Yaskawa INFORM job: DPRINT3D5.JBI

/JOB
//NAME DPRINT3D5
//POS
///NPOS 1005,0,0,0,0,0
///TOOL 9
///POSTYPE PULSE
///PULSE
C00000=38696,60824,-96309,77205,-122166,-85375,0
C00001=38701,60832,-96286,77203,-122174,-85369,0
C00002=38706,60841,-96263,77202,-122182,-85364,0
C00003=38711,60849,-96240,77201,-122190,-85358,0
C00004=38716,60857,-96218,77200,-122199,-85352,0
C00005=38721,60866,-96195,77199,-122207,-85346,0
C00006=38726,60874,-96172,77197,-122215,-85340,0
C00007=38731,60882,-96149,77196,-122223,-85334,0
C00008=38736,60891,-96126,77195,-122232,-85328,0
C00009=38741,60899,-96103,77194,-122240,-85322,0
C00010=38746,60907,-96080,77193,-122248,-85317,0
C00011=38751,60915,-96059,77191,-122256,-85311,0
C00012=38756,60922,-96038,77190,-122264,-85306,0
C00013=38761,60930,-96017,77188,-122272,-85300,0
C00014=38766,60938,-95996,77186,-122280,-85295,0
C00015=38771,60945,-95976,77185,-122289,-85290,0
C00016=38776,60953,-95954,77183,-122297,-85285,0
C00017=38796,60963,-95927,77168,-122315,-85279,0
C00018=38827,60979,-95885,77145,-122344,-85272,0
C00019=38858,60994,-95842,77121,-122374,-85264,0
C00020=38885,61007,-95807,77101,-122398,-85257,0
C00021=38908,61018,-95779,77083,-122418,-85253,0
C00022=38930,61028,-95751,77065,-122439,-85248,0
C00023=38951,61036,-95729,77049,-122456,-85245,0
C00024=38971,61044,-95708,77033,-122474,-85242,0
C00025=38991,61052,-95686,77017,-122491,-85238,0
C00026=39011,61060,-95664,77001,-122509,-85235,0
C00027=39031,61068,-95643,76985,-122526,-85231,0
C00028=39048,61074,-95626,76971,-122540,-85229,0
C00029=39065,61080,-95610,76957,-122555,-85227,0
C00030=39083,61086,-95594,76943,-122570,-85225,0
C00031=39100,61092,-95577,76928,-122584,-85223,0
C00032=39115,61097,-95565,76916,-122597,-85221,0
C00033=39130,61101,-95552,76903,-122609,-85220,0
C00034=39146,61106,-95540,76890,-122622,-85219,0
C00035=39161,61111,-95527,76877,-122633,-85217,0
C00036=39176,61115,-95515,76864,-122646,-85216,0
C00037=39192,61120,-95502,76851,-122659,-85214,0
C00038=39207,61125,-95490,76838,-122671,-85213,0
C00039=39221,61129,-95479,76826,-122683,-85212,0
C00040=39235,61132,-95469,76814,-122693,-85211,0
C00041=39249,61136,-95458,76803,-122705,-85210,0
C00042=39255,61133,-95467,76795,-122706,-85213,0
C00043=39268,61127,-95485,76780,-122710,-85220,0
C00044=39280,61120,-95503,76765,-122714,-85227,0
C00045=39293,61113,-95522,76749,-122717,-85235,0
C00046=39307,61106,-95543,76732,-122721,-85242,0
C00047=39320,61099,-95564,76715,-122724,-85250,0
C00048=39334,61091,-95584,76698,-122728,-85259,0
C00049=39348,61084,-95605,76682,-122732,-85266,0
C00050=39362,61076,-95625,76665,-122736,-85274,0
C00051=39375,61069,-95646,76648,-122739,-85282,0
C00052=39390,61061,-95669,76630,-122742,-85290,0
C00053=39405,61052,-95695,76611,-122746,-85300,0
C00054=39420,61042,-95720,76592,-122749,-85310,0
C00055=39436,61033,-95746,76572,-122753,-85320,0
C00056=39452,61023,-95775,76552,-122756,-85330,0
C00057=39470,61011,-95807,76529,-122760,-85342,0
C00058=39487,61000,-95839,76507,-122763,-85354,0
C00059=39504,60988,-95871,76485,-122765,-85365,0
C00060=39522,60977,-95903,76462,-122769,-85377,0
C00061=39540,60964,-95939,76438,-122772,-85390,0
C00062=39560,60950,-95978,76413,-122775,-85404,0
C00063=39579,60936,-96018,76387,-122777,-85418,0
C00064=39606,60914,-96077,76352,-122779,-85439,0
C00065=39632,60893,-96136,76316,-122782,-85460,0
C00066=39658,60872,-96194,76281,-122784,-85481,0
C00067=39670,60862,-96222,76264,-122785,-85490,0
C00068=39672,60858,-96233,76261,-122783,-85494,0
C00069=39674,60850,-96255,76255,-122779,-85501,0
C00070=39677,60843,-96276,76249,-122776,-85507,0
C00071=39680,60835,-96298,76242,-122772,-85513,0
C00072=39682,60827,-96320,76236,-122769,-85520,0
C00073=39685,60818,-96343,76230,-122764,-85527,0
C00074=39687,60809,-96369,76223,-122761,-85535,0
C00075=39690,60800,-96394,76216,-122756,-85542,0
C00076=39693,60791,-96419,76210,-122752,-85550,0
C00077=39695,60782,-96444,76203,-122747,-85558,0
C00078=39698,60773,-96469,76196,-122742,-85566,0
C00079=39701,60764,-96495,76189,-122738,-85573,0
C00080=39703,60757,-96514,76183,-122736,-85579,0
C00081=39706,60749,-96536,76177,-122732,-85586,0
C00082=39709,60740,-96561,76170,-122728,-85593,0
C00083=39712,60731,-96586,76163,-122723,-85601,0
C00084=39715,60722,-96610,76157,-122719,-85608,0
C00085=39717,60713,-96635,76150,-122715,-85616,0
C00086=39720,60705,-96659,76144,-122710,-85623,0
C00087=39722,60696,-96683,76137,-122706,-85631,0
C00088=39725,60686,-96709,76131,-122701,-85638,0
C00089=39727,60677,-96735,76124,-122696,-85646,0
C00090=39729,60668,-96761,76117,-122692,-85654,0
C00091=39732,60658,-96787,76111,-122687,-85661,0
C00092=39734,60649,-96813,76104,-122683,-85669,0
C00093=39737,60640,-96839,76097,-122678,-85677,0
C00094=39739,60630,-96865,76091,-122674,-85685,0
C00095=39742,60621,-96891,76084,-122669,-85693,0
C00096=39744,60612,-96917,76077,-122663,-85701,0
C00097=39756,60552,-97082,76038,-122631,-85749,0
C00098=39779,60443,-97386,75966,-122571,-85840,0
C00099=39801,60334,-97689,75895,-122511,-85931,0
C00100=37705,58030,-104183,76996,-119736,-87530,0
C00101=42893,55575,-111597,70566,-120383,-90390,0
C00102=44083,55092,-113117,69083,-120456,-90996,0
C00103=26168,57356,-105949,67419,-123808,-89301,0
C00104=27034,56626,-108119,66140,-123522,-90049,0
C00105=31953,53610,-117563,59303,-122121,-93446,0
C00106=30382,53758,-117056,61107,-121729,-93060,0
C00107=38783,58034,-104194,75907,-120329,-87674,0
C00108=39450,58029,-104221,75227,-120689,-87771,0
C00109=39922,58098,-104031,74776,-120996,-87780,0
C00110=45754,54027,-116526,66798,-120045,-92214,0
C00111=45628,53809,-117229,66835,-119751,-92400,0
C00112=45552,53437,-118440,66749,-119301,-92742,0
C00113=45617,53075,-119644,66515,-118904,-93101,0
C00114=45741,52870,-120334,66287,-118707,-93318,0
C00115=31651,54009,-116270,59832,-122529,-93048,0
C00116=31289,54125,-115889,60288,-122540,-92886,0
C00117=30631,54256,-115460,61077,-122448,-92662,0
C00118=30631,54197,-115483,61087,-122475,-92644,0
C00119=46744,53849,-116954,65681,-120330,-92450,0
C00120=46504,53563,-117878,65809,-119907,-92681,0
C00121=46379,53276,-118815,65814,-119525,-92934,0
C00122=46365,52987,-119775,65696,-119175,-93211,0
C00123=46470,52706,-120722,65455,-118871,-93500,0
C00124=46705,52431,-121665,65073,-118611,-93804,0
C00125=31523,53166,-118835,59604,-121482,-93698,0
C00126=31058,53355,-118207,60207,-121566,-93455,0
C00127=30557,53489,-117756,60825,-121555,-93254,0
C00128=30011,53574,-117472,61466,-121459,-93092,0
C00129=29441,53602,-117370,62104,-121278,-92977,0
C00130=28834,53572,-117459,62754,-121010,-92911,0
C00131=24589,59209,-100464,70024,-124680,-87478,0
C00132=24940,59524,-99580,69821,-125135,-87290,0
C00133=25186,59870,-98613,69744,-125558,-87061,0
C00134=25338,60251,-97555,69782,-125954,-86793,0
C00135=25398,60656,-96433,69931,-126315,-86491,0
C00136=29543,55041,-112814,84218,-113592,-89272,0
C00137=37638,58636,-102304,77346,-120164,-86947,0
C00138=38105,58441,-102870,76796,-120296,-87172,0
C00139=38585,58332,-103192,76267,-120488,-87330,0
C00140=39084,58302,-103290,75750,-120742,-87425,0
C00141=39577,58348,-103167,75271,-121047,-87456,0
C00142=40060,58474,-102816,74836,-121406,-87421,0
C00143=46673,53886,-116833,65775,-120344,-92405,0
C00144=47998,53898,-116829,64338,-120877,-92595,0
C00145=47754,53769,-117239,64544,-120631,-92676,0
C00146=47542,53605,-117768,64698,-120356,-92795,0
C00147=47392,53423,-118360,64776,-120082,-92943,0
C00148=47314,53230,-118990,64773,-119821,-93113,0
C00149=47311,53035,-119640,64686,-119581,-93299,0
C00150=47388,52844,-120280,64514,-119373,-93493,0
C00151=47544,52667,-120884,64261,-119205,-93688,0
C00152=47774,52509,-121426,63936,-119085,-93874,0
C00153=47986,52416,-121752,63661,-119035,-93996,0
C00154=31245,52544,-120910,59613,-120533,-94224,0
C00155=31075,52695,-120397,59873,-120683,-94058,0
C00156=30835,52836,-119918,60205,-120793,-93891,0
C00157=30537,52956,-119514,60592,-120849,-93735,0
C00158=30196,53045,-119210,61010,-120845,-93600,0
C00159=29822,53102,-119017,61448,-120783,-93491,0
C00160=29430,53120,-118948,61887,-120665,-93414,0
C00161=29034,53101,-119004,62313,-120495,-93372,0
C00162=28650,53044,-119187,62707,-120280,-93368,0
C00163=28393,52977,-119404,62957,-120101,-93393,0
C00164=23585,59460,-99742,71179,-124323,-87108,0
C00165=23807,59542,-99515,70991,-124513,-87081,0
C00166=24080,59704,-99065,70793,-124797,-86999,0
C00167=24304,59906,-98501,70665,-125087,-86879,0
C00168=24472,60142,-97846,70612,-125369,-86724,0
C00169=24578,60399,-97134,70634,-125635,-86543,0
C00170=24622,60672,-96378,70729,-125875,-86339,0
C00171=24602,60947,-95620,70890,-126076,-86124,0
C00172=24522,61212,-94891,71108,-126232,-85906,0
C00173=24397,61437,-94275,71349,-126328,-85711,0
C00174=37719,59468,-99947,77613,-120758,-86270,0
C00175=37870,59314,-100383,77399,-120746,-86417,0
C00176=38128,59141,-100876,77070,-120782,-86594,0
C00177=38423,59016,-101237,76721,-120867,-86739,0
C00178=38744,58942,-101455,76368,-120999,-86845,0
C00179=39075,58921,-101521,76027,-121174,-86909,0
C00180=39402,58952,-101438,75712,-121381,-86930,0
C00181=39712,59035,-101210,75436,-121615,-86908,0
C00182=39992,59164,-100849,75212,-121866,-86843,0
C00183=40209,59320,-100413,75063,-122100,-86749,0
C00184=47926,53934,-116712,64434,-120891,-92551,0
C00185=48152,53085,-119498,63788,-119950,-93374,0
C00186=48199,52975,-119865,63685,-119829,-93485,0
C00187=48291,52871,-120214,63535,-119731,-93598,0
C00188=48427,52779,-120528,63344,-119660,-93706,0
C00189=48601,52701,-120797,63115,-119621,-93806,0
C00190=48757,52657,-120952,62923,-119617,-93872,0
C00191=48850,52637,-121023,62812,-119622,-93905,0
C00192=49432,52574,-121252,62141,-119740,-94050,0
C00193=30479,51877,-123192,60148,-119327,-94748,0
C00194=30570,52120,-122347,60161,-119708,-94525,0
C00195=30564,52217,-122016,60212,-119842,-94432,0
C00196=30517,52310,-121692,60308,-119958,-94335,0
C00197=30474,52355,-121539,60377,-120006,-94287,0
C00198=30461,52376,-121467,60401,-120032,-94265,0
C00199=30361,52466,-121160,60553,-120121,-94165,0
C00200=30228,52544,-120892,60737,-120183,-94072,0
C00201=30060,52610,-120664,60954,-120215,-93983,0
C00202=29864,52661,-120490,61193,-120215,-93907,0
C00203=29649,52692,-120380,61445,-120182,-93845,0
C00204=29420,52703,-120340,61701,-120115,-93802,0
C00205=29188,52692,-120373,61952,-120018,-93778,0
C00206=28961,52659,-120480,62186,-119894,-93776,0
C00207=28747,52604,-120659,62396,-119747,-93797,0
C00208=28604,52549,-120844,62527,-119622,-93829,0
C00209=28531,52514,-120960,62591,-119551,-93852,0
C00210=28194,52279,-121756,62854,-119121,-94032,0
C00211=22562,59976,-98286,72468,-124138,-86531,0
C00212=22998,59940,-98389,72010,-124363,-86630,0
C00213=23084,59942,-98387,71924,-124413,-86644,0
C00214=23278,59978,-98289,71744,-124554,-86648,0
C00215=23458,60045,-98105,71595,-124709,-86626,0
C00216=23615,60139,-97843,71482,-124874,-86578,0
C00217=23745,60257,-97517,71409,-125040,-86508,0
C00218=23842,60393,-97142,71379,-125202,-86419,0
C00219=23904,60539,-96737,71389,-125351,-86316,0
C00220=23931,60694,-96309,71440,-125485,-86200,0
C00221=23922,60848,-95885,71527,-125597,-86080,0
C00222=23879,60995,-95479,71645,-125683,-85958,0
C00223=23842,61062,-95294,71716,-125712,-85900,0
C00224=23830,61094,-95206,71744,-125729,-85874,0
C00225=23751,61224,-94850,71890,-125777,-85760,0
C00226=23644,61337,-94538,72054,-125798,-85654,0
C00227=23516,61430,-94282,72230,-125788,-85560,0
C00228=23138,61610,-93787,72697,-125688,-85357,0
C00229=38077,60419,-97294,77668,-121580,-85549,0
C00230=38146,60056,-98304,77443,-121390,-85850,0
C00231=38169,59988,-98497,77391,-121360,-85910,0
C00232=38258,59841,-98908,77239,-121319,-86041,0
C00233=38381,59715,-99264,77063,-121308,-86160,0
C00234=38530,59614,-99551,76871,-121330,-86264,0
C00235=38700,59541,-99759,76672,-121381,-86348,0
C00236=38881,59498,-99884,76472,-121458,-86409,0
C00237=39067,59486,-99921,76281,-121558,-86445,0
C00238=39250,59504,-99874,76107,-121676,-86457,0
C00239=39422,59551,-99746,75956,-121808,-86445,0
C00240=39576,59623,-99546,75833,-121947,-86408,0
C00241=39644,59672,-99411,75788,-122020,-86379,0
C00242=39678,59691,-99357,75762,-122053,-86369,0
C00243=39796,59787,-99091,75687,-122187,-86309,0
C00244=39892,59903,-98766,75644,-122324,-86229,0
C00245=39958,60034,-98403,75637,-122453,-86134,0
C00246=40046,60396,-97396,75714,-122752,-85858,0
C00247=49524,53763,-117308,62604,-121298,-92956,0
C00248=49011,53716,-117445,63144,-121047,-92918,0
C00249=48822,53679,-117560,63333,-120931,-92922,0
C00250=48650,53624,-117734,63495,-120799,-92946,0
C00251=48575,53588,-117849,63561,-120727,-92967,0
C00252=48537,53575,-117892,63595,-120697,-92974,0
C00253=48391,53498,-118139,63720,-120549,-93023,0
C00254=48274,53407,-118435,63805,-120394,-93089,0
C00255=48192,53305,-118769,63847,-120237,-93172,0
C00256=48150,53196,-119127,63842,-120088,-93269,0
C00257=48151,53135,-119329,63812,-120012,-93326,0
C00258=47967,53016,-119720,63958,-119797,-93412,0
C00259=49473,53563,-117956,62563,-121031,-93129,0
C00260=49558,53551,-117998,62464,-121049,-93154,0
C00261=49728,53527,-118081,62266,-121081,-93202,0
C00262=49820,53514,-118126,62159,-121098,-93229,0
C00263=49833,53512,-118134,62143,-121100,-93233,0
C00264=49848,53510,-118141,62126,-121103,-93237,0
C00265=49863,53508,-118148,62109,-121106,-93241,0
C00266=49878,53506,-118155,62091,-121110,-93245,0
C00267=49894,53504,-118161,62073,-121112,-93249,0
C00268=49909,53502,-118168,62055,-121115,-93253,0
C00269=49924,53500,-118175,62037,-121119,-93258,0
C00270=49937,53498,-118181,62022,-121121,-93262,0
C00271=49950,53496,-118188,62007,-121123,-93266,0
C00272=49963,53494,-118195,61992,-121126,-93269,0
C00273=49976,53492,-118203,61977,-121128,-93273,0
C00274=49988,53490,-118210,61962,-121129,-93277,0
C00275=50001,53488,-118218,61947,-121130,-93281,0
C00276=50014,53485,-118226,61932,-121132,-93285,0
C00277=50026,53483,-118234,61917,-121134,-93289,0
C00278=50039,53481,-118242,61902,-121136,-93294,0
C00279=50052,53479,-118249,61887,-121137,-93298,0
C00280=50064,53476,-118257,61872,-121139,-93302,0
C00281=50077,53474,-118265,61857,-121141,-93306,0
C00282=50090,53472,-118273,61842,-121143,-93310,0
C00283=50102,53469,-118281,61827,-121144,-93314,0
C00284=50115,53467,-118288,61812,-121146,-93318,0
C00285=50126,53465,-118296,61799,-121147,-93322,0
C00286=50136,53463,-118304,61786,-121149,-93325,0
C00287=50147,53460,-118312,61773,-121150,-93330,0
C00288=50158,53458,-118319,61760,-121150,-93333,0
C00289=50169,53456,-118327,61747,-121151,-93337,0
C00290=50179,53454,-118335,61734,-121152,-93341,0
C00291=50190,53451,-118342,61722,-121153,-93344,0
C00292=50199,53449,-118350,61710,-121153,-93348,0
C00293=50209,53447,-118358,61698,-121154,-93352,0
C00294=50219,53444,-118366,61686,-121154,-93356,0
C00295=50229,53442,-118375,61674,-121155,-93359,0
C00296=50239,53440,-118383,61662,-121155,-93363,0
C00297=50262,53425,-118431,61630,-121146,-93379,0
C00298=50284,53411,-118478,61598,-121136,-93396,0
C00299=50304,53398,-118520,61570,-121127,-93411,0
C00300=50320,53387,-118557,61547,-121118,-93424,0
C00301=50336,53376,-118595,61524,-121110,-93436,0
C00302=50351,53365,-118630,61502,-121101,-93448,0
C00303=50364,53356,-118662,61484,-121093,-93459,0
C00304=50376,53346,-118694,61465,-121085,-93470,0
C00305=50389,53336,-118727,61447,-121077,-93481,0
C00306=50402,53327,-118759,61428,-121069,-93491,0
C00307=50414,53317,-118792,61409,-121061,-93502,0
C00308=50427,53307,-118824,61391,-121053,-93513,0
C00309=50437,53299,-118851,61376,-121045,-93523,0
C00310=50447,53290,-118880,61361,-121038,-93532,0
C00311=50457,53282,-118908,61346,-121030,-93541,0
C00312=50467,53273,-118936,61331,-121023,-93551,0
C00313=50477,53265,-118964,61316,-121015,-93560,0
C00314=50484,53258,-118988,61304,-121010,-93567,0
C00315=50481,53254,-119001,61305,-121004,-93571,0
C00316=50477,53246,-119027,61307,-120991,-93577,0
C00317=50472,53238,-119054,61308,-120979,-93584,0
C00318=50467,53230,-119080,61310,-120967,-93591,0
C00319=50462,53222,-119107,61312,-120954,-93597,0
C00320=50457,53214,-119133,61313,-120942,-93604,0
C00321=50452,53206,-119159,61315,-120930,-93610,0
C00322=50447,53198,-119186,61317,-120918,-93617,0
C00323=50442,53190,-119212,61318,-120905,-93624,0
C00324=50436,53182,-119240,61321,-120892,-93630,0
C00325=50429,53173,-119267,61324,-120879,-93637,0
C00326=50423,53165,-119296,61327,-120866,-93644,0
C00327=50417,53156,-119324,61329,-120852,-93651,0
C00328=50411,53148,-119351,61332,-120839,-93658,0
C00329=50403,53138,-119383,61337,-120823,-93665,0
C00330=50394,53128,-119416,61341,-120807,-93673,0
C00331=50386,53118,-119448,61346,-120792,-93681,0
C00332=50378,53109,-119480,61350,-120776,-93689,0
C00333=50369,53099,-119512,61355,-120760,-93696,0
C00334=50361,53089,-119544,61359,-120745,-93704,0
C00335=50353,53080,-119575,61364,-120729,-93711,0
C00336=50343,53070,-119610,61369,-120713,-93719,0
C00337=50333,53059,-119645,61376,-120695,-93728,0
C00338=50322,53048,-119681,61382,-120676,-93736,0
C00339=50309,53036,-119721,61391,-120656,-93746,0
C00340=50294,53022,-119766,61401,-120633,-93756,0
C00341=50279,53008,-119812,61412,-120608,-93766,0
C00342=50263,52995,-119858,61422,-120585,-93777,0
C00343=50248,52981,-119903,61432,-120563,-93787,0
C00344=50229,52965,-119955,61445,-120535,-93799,0
C00345=50208,52948,-120011,61461,-120505,-93812,0
C00346=50177,52927,-120083,61485,-120466,-93827,0
C00347=50147,52905,-120155,61508,-120426,-93843,0
C00348=50117,52883,-120226,61531,-120387,-93859,0
C00349=50037,52836,-120384,61596,-120296,-93891,0
C00350=50025,52833,-120391,61609,-120289,-93892,0
C00351=50012,52831,-120398,61622,-120282,-93892,0
C00352=50000,52829,-120404,61634,-120275,-93892,0
C00353=49988,52827,-120411,61647,-120268,-93892,0
C00354=49976,52825,-120418,61659,-120261,-93892,0
C00355=49963,52823,-120425,61672,-120255,-93892,0
C00356=49951,52821,-120430,61684,-120248,-93892,0
C00357=49939,52819,-120437,61697,-120240,-93892,0
C00358=49869,52809,-120469,61770,-120202,-93891,0
C00359=49740,52791,-120528,61902,-120134,-93889,0
C00360=49612,52773,-120584,62036,-120066,-93887,0
C00361=49483,52755,-120642,62169,-119997,-93885,0
C00362=30116,51956,-122908,60587,-119324,-94619,0
C00363=30009,51889,-123144,60673,-119192,-94671,0
C00364=29902,51821,-123378,60760,-119059,-94722,0
C00365=29894,51816,-123395,60767,-119050,-94726,0
C00366=29885,51811,-123411,60775,-119040,-94729,0
C00367=29876,51806,-123431,60782,-119030,-94734,0
C00368=29867,51799,-123453,60790,-119017,-94738,0
C00369=29857,51793,-123474,60797,-119004,-94743,0
C00370=29847,51787,-123496,60805,-118993,-94748,0
C00371=29838,51781,-123518,60813,-118980,-94753,0
C00372=29828,51775,-123540,60821,-118969,-94758,0
C00373=29820,51770,-123557,60828,-118958,-94762,0
C00374=29811,51764,-123574,60835,-118948,-94766,0
C00375=29802,51759,-123593,60843,-118938,-94769,0
C00376=29793,51754,-123610,60850,-118928,-94773,0
C00377=29784,51750,-123626,60858,-118918,-94777,0
C00378=29775,51745,-123643,60866,-118908,-94780,0
C00379=29766,51740,-123661,60874,-118899,-94784,0
C00380=29757,51735,-123677,60882,-118888,-94787,0
C00381=29748,51730,-123694,60890,-118879,-94791,0
C00382=29738,51726,-123710,60898,-118869,-94794,0
C00383=29729,51721,-123727,60906,-118858,-94798,0
C00384=29720,51716,-123745,60914,-118849,-94801,0
C00385=29711,51711,-123761,60922,-118839,-94805,0
C00386=29701,51706,-123778,60930,-118828,-94808,0
C00387=29692,51702,-123794,60938,-118819,-94812,0
C00388=29684,51698,-123809,60945,-118810,-94814,0
C00389=29675,51694,-123823,60953,-118802,-94817,0
C00390=29667,51690,-123836,60960,-118794,-94820,0
C00391=29658,51686,-123850,60968,-118785,-94823,0
C00392=29650,51682,-123864,60975,-118777,-94826,0
C00393=29642,51678,-123878,60983,-118768,-94828,0
C00394=29633,51674,-123890,60990,-118759,-94831,0
C00395=29625,51671,-123903,60998,-118753,-94834,0
C00396=29617,51667,-123916,61005,-118745,-94836,0
C00397=29608,51663,-123927,61013,-118736,-94838,0
C00398=29600,51660,-123940,61021,-118728,-94841,0
C00399=29592,51656,-123953,61028,-118722,-94843,0
C00400=29555,51651,-123971,61066,-118701,-94843,0
C00401=29519,51645,-123990,61104,-118681,-94844,0
C00402=29486,51641,-124005,61137,-118664,-94845,0
C00403=29458,51637,-124018,61167,-118650,-94844,0
C00404=29430,51634,-124030,61196,-118637,-94844,0
C00405=29405,51631,-124040,61223,-118624,-94843,0
C00406=29381,51628,-124048,61248,-118612,-94843,0
C00407=29358,51626,-124056,61273,-118602,-94842,0
C00408=29334,51623,-124064,61298,-118591,-94841,0
C00409=29311,51621,-124072,61323,-118580,-94841,0
C00410=29287,51619,-124081,61347,-118569,-94840,0
C00411=29264,51616,-124089,61372,-118557,-94839,0
C00412=29243,51614,-124094,61394,-118549,-94838,0
C00413=29223,51613,-124100,61416,-118540,-94836,0
C00414=29202,51611,-124105,61438,-118531,-94835,0
C00415=29181,51610,-124111,61460,-118522,-94835,0
C00416=29161,51608,-124116,61482,-118512,-94834,0
C00417=29148,51607,-124118,61496,-118508,-94832,0
C00418=29142,51607,-124119,61503,-118506,-94832,0
C00419=29128,51611,-124103,61520,-118508,-94825,0
C00420=29114,51616,-124087,61537,-118509,-94819,0
C00421=29100,51620,-124070,61554,-118511,-94813,0
C00422=29087,51625,-124054,61572,-118514,-94806,0
C00423=29073,51630,-124038,61589,-118516,-94799,0
C00424=29059,51634,-124020,61606,-118518,-94793,0
C00425=29046,51639,-124004,61623,-118520,-94787,0
C00426=29032,51643,-123988,61640,-118523,-94780,0
C00427=29018,51648,-123970,61658,-118525,-94773,0
C00428=29004,51654,-123951,61676,-118529,-94766,0
C00429=28989,51659,-123932,61694,-118531,-94759,0
C00430=28975,51664,-123912,61713,-118534,-94751,0
C00431=28961,51670,-123894,61731,-118537,-94744,0
C00432=28946,51675,-123872,61750,-118541,-94736,0
C00433=28930,51682,-123849,61771,-118545,-94727,0
C00434=28914,51689,-123825,61791,-118549,-94718,0
C00435=28898,51695,-123802,61812,-118554,-94709,0
C00436=28882,51702,-123778,61832,-118557,-94701,0
C00437=28867,51708,-123755,61852,-118562,-94692,0
C00438=28851,51715,-123731,61873,-118566,-94683,0
C00439=28835,51722,-123708,61893,-118570,-94675,0
C00440=28818,51729,-123679,61916,-118576,-94664,0
C00441=28801,51737,-123651,61938,-118581,-94654,0
C00442=28784,51745,-123623,61960,-118587,-94644,0
C00443=28763,51756,-123585,61989,-118595,-94630,0
C00444=28742,51767,-123546,62017,-118604,-94616,0
C00445=28720,51778,-123507,62045,-118612,-94602,0
C00446=28699,51789,-123468,62073,-118620,-94588,0
C00447=28678,51800,-123428,62102,-118630,-94574,0
C00448=28653,51815,-123377,62137,-118641,-94556,0
C00449=28624,51832,-123315,62176,-118656,-94535,0
C00450=28593,51852,-123245,62219,-118674,-94510,0
C00451=28563,51872,-123175,62262,-118692,-94487,0
C00452=28517,51904,-123062,62327,-118720,-94448,0
C00453=28483,51931,-122964,62376,-118748,-94416,0
C00454=28484,51934,-122954,62377,-118753,-94413,0
C00455=28484,51940,-122933,62379,-118761,-94407,0
C00456=28485,51946,-122913,62381,-118769,-94401,0
C00457=28486,51952,-122892,62383,-118778,-94395,0
C00458=28486,51958,-122871,62385,-118786,-94390,0
C00459=28487,51964,-122850,62387,-118794,-94384,0
C00460=28487,51970,-122831,62389,-118802,-94378,0
C00461=28488,51976,-122810,62391,-118811,-94372,0
C00462=28488,51982,-122790,62394,-118819,-94366,0
C00463=28502,52043,-122577,62407,-118908,-94308,0
C00464=28514,52104,-122364,62421,-118995,-94249,0
C00465=28527,52166,-122152,62435,-119084,-94190,0
C00466=28533,52197,-122046,62442,-119127,-94160,0
C00467=22674,60229,-97582,72478,-124393,-86349,0
C00468=22555,60286,-97421,72625,-124366,-86285,0
C00469=22432,60347,-97251,72779,-124339,-86217,0
C00470=22422,60353,-97235,72792,-124337,-86211,0
C00471=22411,60358,-97220,72805,-124335,-86205,0
C00472=22400,60364,-97204,72819,-124333,-86199,0
C00473=22390,60369,-97189,72832,-124331,-86193,0
C00474=22379,60375,-97173,72845,-124328,-86186,0
C00475=22369,60381,-97158,72859,-124326,-86180,0
C00476=22358,60386,-97142,72872,-124324,-86174,0
C00477=22348,60392,-97126,72885,-124321,-86168,0
C00478=22338,60397,-97111,72898,-124320,-86162,0
C00479=22329,60402,-97096,72909,-124319,-86157,0
C00480=22320,60408,-97082,72921,-124318,-86151,0
C00481=22311,60413,-97067,72932,-124316,-86145,0
C00482=22303,60419,-97051,72943,-124316,-86139,0
C00483=22294,60424,-97036,72954,-124314,-86134,0
C00484=22286,60429,-97021,72965,-124313,-86128,0
C00485=22278,60435,-97006,72976,-124312,-86123,0
C00486=22270,60440,-96991,72987,-124311,-86117,0
C00487=22261,60446,-96976,72998,-124311,-86112,0
C00488=22253,60451,-96961,73009,-124310,-86106,0
C00489=22245,60457,-96945,73020,-124309,-86101,0
C00490=22241,60459,-96938,73025,-124309,-86098,0
C00491=22220,60506,-96808,73069,-124331,-86058,0
C00492=22199,60561,-96656,73116,-124358,-86011,0
C00493=22188,60597,-96555,73145,-124378,-85980,0
C00494=22176,60634,-96454,73174,-124397,-85950,0
C00495=22167,60666,-96365,73199,-124416,-85924,0
C00496=22159,60694,-96289,73220,-124431,-85901,0
C00497=22155,60716,-96227,73235,-124444,-85882,0
C00498=22151,60739,-96165,73251,-124458,-85864,0
C00499=22146,60761,-96102,73266,-124472,-85846,0
C00500=22142,60784,-96040,73282,-124486,-85828,0
C00501=22137,60806,-95978,73297,-124500,-85809,0
C00502=22135,60823,-95932,73307,-124510,-85796,0
C00503=22133,60840,-95885,73318,-124520,-85783,0
C00504=22130,60857,-95839,73328,-124532,-85769,0
C00505=22129,60872,-95797,73337,-124541,-85757,0
C00506=22128,60887,-95755,73346,-124551,-85745,0
C00507=22126,60903,-95713,73354,-124562,-85733,0
C00508=22125,60918,-95671,73363,-124572,-85720,0
C00509=22124,60933,-95629,73372,-124582,-85708,0
C00510=22123,60948,-95587,73380,-124593,-85696,0
C00511=22122,60964,-95544,73389,-124603,-85684,0
C00512=22121,60978,-95506,73397,-124612,-85673,0
C00513=22121,60991,-95470,73403,-124621,-85663,0
C00514=22120,61003,-95435,73410,-124631,-85653,0
C00515=22120,61016,-95400,73416,-124640,-85643,0
C00516=22120,61029,-95364,73423,-124649,-85633,0
C00517=22120,61042,-95329,73429,-124658,-85623,0
C00518=22120,61054,-95296,73434,-124667,-85614,0
C00519=22121,61066,-95262,73440,-124675,-85604,0
C00520=22121,61079,-95228,73446,-124685,-85595,0
C00521=22121,61091,-95194,73451,-124694,-85585,0
C00522=22122,61104,-95160,73457,-124703,-85575,0
C00523=22122,61116,-95126,73463,-124712,-85566,0
C00524=22123,61128,-95093,73468,-124721,-85557,0
C00525=22123,61140,-95059,73474,-124730,-85547,0
C00526=22133,61149,-95035,73468,-124742,-85542,0
C00527=22145,61158,-95010,73460,-124757,-85537,0
C00528=22158,61168,-94984,73453,-124771,-85532,0
C00529=22170,61177,-94959,73445,-124785,-85527,0
C00530=22182,61186,-94933,73438,-124798,-85521,0
C00531=22194,61196,-94908,73430,-124812,-85516,0
C00532=22209,61206,-94880,73421,-124829,-85510,0
C00533=22224,61217,-94851,73411,-124845,-85505,0
C00534=22239,61227,-94823,73401,-124863,-85499,0
C00535=22254,61237,-94795,73392,-124879,-85494,0
C00536=22269,61248,-94766,73382,-124895,-85488,0
C00537=22283,61258,-94738,73372,-124912,-85483,0
C00538=22300,61269,-94708,73361,-124930,-85477,0
C00539=22318,61281,-94677,73349,-124949,-85471,0
C00540=22336,61292,-94645,73336,-124968,-85465,0
C00541=22357,61305,-94612,73322,-124990,-85459,0
C00542=22380,61318,-94577,73306,-125013,-85452,0
C00543=22402,61331,-94541,73290,-125036,-85447,0
C00544=22414,61337,-94523,73281,-125048,-85443,0
C00545=22418,61338,-94522,73277,-125051,-85444,0
C00546=22427,61339,-94519,73269,-125057,-85444,0
C00547=22435,61340,-94517,73261,-125063,-85445,0
C00548=22444,61341,-94514,73253,-125068,-85445,0
C00549=22453,61342,-94512,73245,-125075,-85447,0
C00550=22462,61342,-94510,73237,-125081,-85447,0
C00551=22471,61343,-94508,73228,-125087,-85448,0
C00552=22480,61344,-94506,73218,-125094,-85449,0
C00553=22490,61344,-94504,73209,-125099,-85451,0
C00554=22500,61345,-94503,73200,-125106,-85452,0
C00555=22509,61346,-94501,73191,-125112,-85453,0
C00556=22518,61346,-94499,73182,-125119,-85454,0
C00557=22529,61347,-94499,73171,-125126,-85455,0
C00558=22540,61347,-94498,73161,-125133,-85457,0
C00559=22551,61347,-94498,73150,-125138,-85459,0
C00560=22561,61348,-94497,73140,-125145,-85460,0
C00561=22572,61348,-94496,73129,-125152,-85462,0
C00562=22583,61348,-94496,73119,-125159,-85463,0
C00563=22594,61348,-94495,73108,-125166,-85465,0
C00564=22604,61349,-94494,73098,-125173,-85466,0
C00565=22615,61349,-94494,73087,-125180,-85468,0
C00566=22626,61349,-94493,73077,-125187,-85470,0
C00567=22637,61349,-94492,73066,-125194,-85472,0
C00568=22647,61350,-94492,73056,-125199,-85473,0
C00569=22658,61349,-94493,73044,-125206,-85475,0
C00570=22669,61349,-94493,73033,-125213,-85477,0
C00571=22680,61349,-94494,73023,-125220,-85479,0
C00572=22692,61349,-94495,73010,-125227,-85481,0
C00573=22706,61348,-94498,72997,-125234,-85484,0
C00574=22719,61347,-94500,72983,-125242,-85487,0
C00575=22732,61346,-94503,72970,-125249,-85490,0
C00576=22745,61345,-94505,72956,-125257,-85493,0
C00577=22758,61344,-94508,72942,-125264,-85496,0
C00578=22772,61344,-94510,72929,-125272,-85499,0
C00579=22785,61343,-94512,72915,-125279,-85502,0
C00580=22798,61342,-94515,72902,-125287,-85505,0
C00581=22810,61341,-94518,72889,-125294,-85508,0
C00582=22822,61340,-94521,72877,-125299,-85510,0
C00583=22907,61327,-94557,72786,-125342,-85535,0
C00584=23065,61303,-94624,72616,-125421,-85580,0
C00585=38394,60398,-97360,77346,-121758,-85612,0
C00586=38429,60511,-97047,77361,-121851,-85527,0
C00587=38465,60629,-96720,77378,-121948,-85437,0
C00588=38469,60639,-96691,77379,-121956,-85429,0
C00589=38472,60650,-96663,77380,-121966,-85422,0
C00590=38476,60660,-96634,77381,-121975,-85414,0
C00591=38479,60670,-96606,77382,-121983,-85406,0
C00592=38483,60681,-96577,77383,-121992,-85398,0
C00593=38486,60691,-96549,77385,-122000,-85391,0
C00594=38490,60701,-96520,77386,-122009,-85383,0
C00595=38493,60712,-96492,77387,-122017,-85375,0
C00596=38497,60721,-96465,77388,-122025,-85368,0
C00597=38500,60730,-96440,77388,-122033,-85361,0
C00598=38504,60739,-96416,77389,-122041,-85355,0
C00599=38507,60748,-96391,77389,-122050,-85348,0
C00600=38511,60757,-96368,77389,-122058,-85342,0
C00601=38515,60765,-96345,77389,-122064,-85336,0
C00602=38519,60773,-96321,77389,-122072,-85330,0
C00603=38523,60782,-96298,77389,-122081,-85324,0
C00604=38527,60790,-96275,77389,-122087,-85318,0
C00605=38530,60799,-96252,77389,-122095,-85311,0
C00606=38534,60807,-96229,77389,-122104,-85306,0
C00607=38538,60815,-96206,77388,-122110,-85299,0
C00608=38540,60820,-96194,77389,-122115,-85296,0
C00609=38587,60851,-96109,77357,-122163,-85278,0
C00610=38642,60883,-96021,77317,-122217,-85260,0
C00611=38679,60904,-95965,77290,-122253,-85250,0
C00612=38716,60924,-95910,77262,-122289,-85239,0
C00613=38749,60941,-95863,77238,-122320,-85230,0
C00614=38778,60955,-95825,77216,-122347,-85223,0
C00615=38801,60966,-95797,77198,-122368,-85219,0
C00616=38825,60976,-95769,77179,-122389,-85214,0
C00617=38848,60986,-95741,77161,-122409,-85209,0
C00618=38871,60997,-95713,77143,-122431,-85205,0
C00619=38895,61007,-95685,77124,-122452,-85200,0
C00620=38913,61014,-95667,77110,-122467,-85197,0
C00621=38930,61021,-95648,77096,-122482,-85194,0
C00622=38948,61027,-95630,77082,-122498,-85192,0
C00623=38964,61033,-95615,77068,-122510,-85190,0
C00624=38981,61038,-95600,77055,-122524,-85188,0
C00625=38997,61044,-95585,77041,-122538,-85185,0
C00626=39013,61049,-95570,77028,-122552,-85184,0
C00627=39029,61055,-95556,77014,-122565,-85182,0
C00628=39046,61061,-95541,77001,-122579,-85180,0
C00629=39062,61066,-95526,76987,-122592,-85178,0
C00630=39077,61071,-95513,76975,-122605,-85177,0
C00631=39091,61075,-95502,76963,-122616,-85176,0
C00632=39105,61079,-95491,76951,-122626,-85174,0
C00633=39119,61083,-95480,76940,-122638,-85173,0
C00634=39132,61087,-95470,76928,-122649,-85172,0
C00635=39146,61091,-95460,76916,-122660,-85171,0
C00636=39160,61094,-95451,76905,-122670,-85170,0
C00637=39173,61097,-95442,76893,-122680,-85170,0
C00638=39186,61100,-95434,76881,-122691,-85169,0
C00639=39200,61104,-95425,76870,-122701,-85169,0
C00640=39213,61107,-95416,76858,-122711,-85168,0
C00641=39227,61110,-95407,76846,-122722,-85167,0
C00642=39240,61114,-95398,76835,-122732,-85167,0
C00643=39253,61117,-95390,76823,-122742,-85166,0
C00644=39265,61111,-95407,76809,-122746,-85173,0
C00645=39279,61103,-95428,76792,-122749,-85181,0
C00646=39292,61096,-95449,76775,-122753,-85189,0
C00647=39306,61088,-95470,76759,-122757,-85197,0
C00648=39319,61081,-95491,76742,-122761,-85205,0
C00649=39333,61073,-95512,76726,-122764,-85213,0
C00650=39348,61063,-95538,76706,-122767,-85223,0
C00651=39364,61054,-95565,76687,-122770,-85233,0
C00652=39379,61044,-95592,76667,-122773,-85243,0
C00653=39394,61035,-95619,76648,-122777,-85253,0
C00654=39410,61025,-95645,76628,-122780,-85263,0
C00655=39425,61015,-95672,76609,-122784,-85273,0
C00656=39442,61005,-95702,76588,-122787,-85284,0
C00657=39459,60993,-95736,76565,-122790,-85296,0
C00658=39477,60981,-95769,76542,-122793,-85308,0
C00659=39496,60967,-95808,76517,-122795,-85322,0
C00660=39516,60951,-95851,76490,-122798,-85337,0
C00661=39537,60936,-95894,76463,-122800,-85353,0
C00662=39547,60928,-95916,76449,-122801,-85360,0
C00663=39549,60924,-95926,76446,-122800,-85363,0
C00664=39552,60917,-95945,76440,-122798,-85369,0
C00665=39556,60910,-95964,76433,-122795,-85375,0
C00666=39559,60903,-95983,76426,-122793,-85382,0
C00667=39563,60896,-96003,76420,-122791,-85387,0
C00668=39566,60889,-96023,76413,-122788,-85394,0
C00669=39570,60881,-96045,76406,-122785,-85401,0
C00670=39573,60873,-96067,76399,-122782,-85407,0
C00671=39577,60865,-96088,76392,-122779,-85414,0
C00672=39580,60857,-96110,76385,-122776,-85421,0
C00673=39584,60850,-96132,76378,-122772,-85427,0
C00674=39587,60842,-96154,76371,-122770,-85434,0
C00675=39590,60833,-96179,76364,-122765,-85442,0
C00676=39594,60823,-96205,76356,-122762,-85450,0
C00677=39597,60814,-96230,76349,-122757,-85458,0
C00678=39601,60805,-96255,76341,-122754,-85466,0
C00679=39604,60796,-96281,76334,-122750,-85473,0
C00680=39607,60787,-96306,76326,-122746,-85481,0
C00681=39611,60777,-96332,76318,-122742,-85489,0
C00682=39614,60768,-96357,76311,-122738,-85496,0
C00683=39618,60759,-96382,76303,-122734,-85505,0
C00684=39621,60750,-96408,76296,-122731,-85512,0
C00685=39624,60741,-96433,76288,-122726,-85520,0
C00686=39628,60732,-96458,76281,-122723,-85528,0
C00687=39630,60723,-96484,76274,-122718,-85535,0
C00688=39633,60713,-96509,76267,-122714,-85543,0
C00689=39636,60704,-96534,76260,-122709,-85550,0
C00690=39639,60694,-96564,76253,-122705,-85560,0
C00691=39642,60682,-96595,76245,-122699,-85569,0
C00692=39644,60671,-96625,76237,-122693,-85578,0
C00693=39647,60661,-96656,76229,-122687,-85587,0
C00694=39650,60650,-96686,76222,-122682,-85596,0
C00695=39653,60639,-96716,76214,-122676,-85605,0
C00696=39656,60628,-96746,76206,-122671,-85614,0
C00697=39658,60617,-96777,76199,-122665,-85624,0
C00698=39661,60606,-96807,76191,-122660,-85633,0
C00699=39664,60595,-96837,76184,-122654,-85642,0
C00700=39666,60585,-96865,76177,-122648,-85650,0
C00701=39676,60510,-97073,76133,-122605,-85711,0
C00702=39694,60371,-97458,76052,-122524,-85824,0
C00703=37498,58093,-103859,77262,-119719,-87384,0
C00704=42894,55517,-111620,70575,-120403,-90371,0
C00705=44083,55033,-113140,69092,-120477,-90977,0
C00706=26168,57300,-105971,67430,-123828,-89283,0
C00707=27034,56569,-108141,66150,-123543,-90031,0
C00708=31954,53550,-117586,59313,-122149,-93427,0
C00709=30399,53730,-116974,61115,-121804,-93014,0
C00710=38797,58060,-103981,75937,-120411,-87588,0
C00711=39143,58040,-104047,75577,-120585,-87653,0
C00712=39793,58101,-103882,74944,-120985,-87693,0
C00713=39843,58114,-103846,74898,-121022,-87690,0
C00714=45706,53993,-116462,66873,-120079,-92163,0
C00715=45675,53958,-116576,66890,-120027,-92192,0
C00716=45503,53576,-117808,66902,-119533,-92525,0
C00717=45474,53191,-119072,66760,-119082,-92888,0
C00718=45598,52819,-120315,66457,-118692,-93268,0
C00719=45645,52761,-120513,66380,-118639,-93331,0
C00720=31712,53968,-116230,59786,-122605,-93022,0
C00721=31655,53993,-116152,59860,-122614,-92992,0
C00722=31009,54173,-115565,60660,-122593,-92727,0
C00723=30647,54230,-115376,61086,-122523,-92618,0
C00724=30647,54171,-115398,61096,-122549,-92598,0
C00725=46650,53838,-116817,65815,-120373,-92371,0
C00726=46480,53664,-117375,65920,-120109,-92507,0
C00727=46314,53371,-118323,65966,-119706,-92757,0
C00728=46258,53074,-119302,65890,-119338,-93032,0
C00729=46319,52783,-120271,65693,-119012,-93321,0
C00730=46427,52615,-120841,65498,-118847,-93501,0
C00731=46674,52353,-121739,65109,-118607,-93794,0
C00732=31639,53141,-118742,59503,-121600,-93666,0
C00733=31365,53267,-118323,59866,-121669,-93509,0
C00734=30867,53422,-117808,60490,-121690,-93291,0
C00735=30324,53526,-117459,61138,-121621,-93111,0
C00736=29754,53576,-117287,61787,-121467,-92977,0
C00737=29399,53571,-117297,62174,-121326,-92925,0
C00738=28814,53531,-117416,62796,-121052,-92870,0
C00739=24540,59243,-100236,70130,-124744,-87381,0
C00740=24732,59379,-99857,70000,-124963,-87308,0
C00741=25016,59681,-99013,69860,-125369,-87120,0
C00742=25219,60027,-98051,69828,-125766,-86887,0
C00743=25335,60404,-97006,69903,-126137,-86616,0
C00744=29566,54807,-113384,84149,-113515,-89424,0
C00745=29507,54971,-112873,84257,-113580,-89260,0
C00746=37737,58639,-102164,77280,-120274,-86893,0
C00747=37947,58523,-102498,77022,-120314,-87018,0
C00748=38381,58376,-102928,76524,-120458,-87200,0
C00749=38847,58299,-103157,76022,-120664,-87329,0
C00750=39325,58296,-103177,75537,-120927,-87399,0
C00751=39796,58365,-102987,75090,-121237,-87409,0
C00752=40037,58441,-102774,74879,-121426,-87381,0
C00753=46579,53874,-116697,65909,-120387,-92327,0
C00754=47885,53894,-116667,64498,-120924,-92507,0
C00755=47602,53736,-117170,64731,-120630,-92608,0
C00756=47485,53640,-117479,64814,-120472,-92679,0
C00757=47343,53492,-117957,64900,-120242,-92795,0
C00758=47234,53292,-118609,64926,-119964,-92966,0
C00759=47203,53088,-119280,64866,-119706,-93154,0
C00760=47251,52888,-119945,64722,-119481,-93352,0
C00761=47319,52787,-120287,64601,-119380,-93459,0
C00762=47454,52645,-120766,64388,-119251,-93615,0
C00763=47696,52489,-121303,64051,-119139,-93802,0
C00764=48003,52362,-121746,63655,-119080,-93970,0
C00765=31385,52522,-120799,59488,-120665,-94189,0
C00766=31176,52697,-120207,59802,-120835,-93995,0
C00767=31031,52778,-119934,60000,-120895,-93899,0
C00768=30796,52884,-119574,60310,-120956,-93765,0
C00769=30452,52989,-119219,60740,-120973,-93616,0
C00770=30075,53060,-118979,61189,-120929,-93493,0
C00771=29678,53094,-118861,61642,-120827,-93401,0
C00772=29460,53091,-118866,61879,-120744,-93370,0
C00773=29143,53070,-118931,62217,-120599,-93342,0
C00774=28759,53005,-119136,62608,-120375,-93343,0
C00775=28405,52905,-119463,62949,-120118,-93385,0
C00776=23544,59484,-99546,71269,-124380,-87022,0
C00777=23924,59657,-99067,70966,-124732,-86949,0
C00778=24159,59823,-98605,70809,-124998,-86860,0
C00779=24349,60026,-98042,70717,-125267,-86734,0
C00780=24487,60257,-97401,70694,-125529,-86578,0
C00781=24568,60509,-96705,70739,-125774,-86397,0
C00782=24589,60772,-95979,70852,-125992,-86198,0
C00783=24552,61037,-95249,71026,-126174,-85987,0
C00784=24537,61078,-95138,71062,-126196,-85954,0
C00785=24517,61177,-94866,71133,-126260,-85874,0
C00786=24421,61394,-94271,71342,-126366,-85691,0
C00787=37804,59465,-99826,77561,-120856,-86221,0
C00788=38099,59210,-100550,77159,-120861,-86471,0
C00789=38353,59067,-100959,76845,-120913,-86624,0
C00790=38639,58968,-101246,76517,-121011,-86745,0
C00791=38946,58916,-101398,76188,-121151,-86831,0
C00792=39260,58914,-101412,75872,-121328,-86878,0
C00793=39569,58961,-101285,75581,-121536,-86884,0
C00794=39862,59055,-101023,75329,-121769,-86850,0
C00795=39903,59077,-100961,75297,-121808,-86838,0
C00796=40008,59117,-100851,75209,-121897,-86821,0
C00797=40227,59249,-100483,75048,-122115,-86746,0
C00798=47813,53930,-116550,64594,-120938,-92463,0
C00799=48076,52988,-119634,63864,-119905,-93376,0
C00800=48105,52947,-119773,63813,-119864,-93419,0
C00801=48187,52862,-120059,63684,-119787,-93512,0
C00802=48330,52770,-120372,63484,-119720,-93621,0
C00803=48507,52696,-120627,63255,-119688,-93718,0
C00804=48710,52641,-120815,63007,-119688,-93800,0
C00805=48929,52609,-120933,62751,-119722,-93863,0
C00806=49558,52580,-121047,62043,-119902,-93983,0
C00807=30639,51856,-123072,60000,-119469,-94711,0
C00808=30695,52140,-122087,60071,-119896,-94444,0
C00809=30668,52250,-121711,60152,-120042,-94336,0
C00810=30595,52357,-121344,60283,-120166,-94224,0
C00811=30477,52457,-121001,60461,-120264,-94112,0
C00812=30418,52490,-120890,60542,-120289,-94072,0
C00813=30277,52553,-120674,60727,-120326,-93992,0
C00814=30072,52615,-120463,60982,-120337,-93903,0
C00815=29846,52656,-120319,61250,-120313,-93831,0
C00816=29607,52676,-120249,61522,-120256,-93777,0
C00817=29517,52675,-120251,61621,-120222,-93765,0
C00818=29325,52662,-120290,61826,-120137,-93748,0
C00819=29097,52624,-120412,62059,-120006,-93750,0
C00820=28891,52567,-120602,62259,-119857,-93774,0
C00821=28713,52493,-120847,62419,-119697,-93819,0
C00822=28572,52407,-121137,62535,-119533,-93881,0
C00823=28282,52139,-122046,62731,-119075,-94101,0
C00824=22501,60048,-97956,72601,-124213,-86403,0
C00825=22918,59992,-98119,72153,-124413,-86517,0
C00826=23094,59998,-98103,71978,-124521,-86541,0
C00827=23258,60033,-98009,71829,-124643,-86542,0
C00828=23288,60044,-97977,71804,-124670,-86537,0
C00829=23382,60070,-97907,71722,-124743,-86533,0
C00830=23528,60137,-97722,71608,-124880,-86506,0
C00831=23657,60230,-97466,71523,-125026,-86455,0
C00832=23762,60342,-97155,71472,-125174,-86385,0
C00833=23840,60471,-96801,71458,-125318,-86299,0
C00834=23886,60610,-96416,71482,-125452,-86199,0
C00835=23900,60756,-96015,71541,-125572,-86089,0
C00836=23881,60902,-95613,71634,-125671,-85973,0
C00837=23872,60927,-95544,71655,-125684,-85952,0
C00838=23857,61008,-95320,71712,-125736,-85886,0
C00839=23794,61153,-94923,71849,-125807,-85764,0
C00840=23702,61283,-94565,72007,-125849,-85648,0
C00841=23580,61398,-94250,72188,-125859,-85538,0
C00842=23258,61604,-93685,72613,-125812,-85325,0
C00843=38206,60451,-97084,77588,-121725,-85481,0
C00844=38247,60096,-98070,77393,-121524,-85772,0
C00845=38299,59955,-98464,77281,-121466,-85893,0
C00846=38380,59832,-98808,77148,-121434,-86004,0
C00847=38400,59812,-98866,77119,-121432,-86023,0
C00848=38451,59745,-99055,77039,-121420,-86085,0
C00849=38568,59644,-99340,76880,-121422,-86184,0
C00850=38708,59564,-99566,76707,-121451,-86268,0
C00851=38864,59509,-99724,76527,-121506,-86336,0
C00852=39032,59480,-99808,76347,-121584,-86383,0
C00853=39203,59478,-99816,76176,-121683,-86409,0
C00854=39372,59505,-99746,76019,-121799,-86413,0
C00855=39532,59557,-99601,75883,-121929,-86394,0
C00856=39557,59571,-99563,75863,-121953,-86386,0
C00857=39644,59604,-99471,75792,-122025,-86372,0
C00858=39787,59692,-99229,75688,-122169,-86323,0
C00859=39907,59803,-98920,75618,-122316,-86251,0
C00860=39999,59934,-98556,75586,-122460,-86160,0
C00861=40130,60257,-97660,75602,-122757,-85922,0
C00862=49395,53762,-117135,62784,-121349,-92862,0
C00863=48813,53686,-117364,63385,-121035,-92840,0
C00864=48604,53635,-117524,63590,-120895,-92854,0
C00865=48415,53563,-117752,63763,-120736,-92890,0
C00866=48252,53473,-118042,63898,-120565,-92949,0
C00867=48204,53433,-118170,63932,-120499,-92978,0
C00868=48121,53345,-118456,63982,-120361,-93048,0
C00869=48060,53227,-118842,63994,-120194,-93148,0
C00870=48044,53107,-119240,63954,-120041,-93259,0
C00871=48062,53039,-119466,63903,-119963,-93326,0
C00872=48011,52957,-119735,63922,-119843,-93396,0
C00873=49351,53558,-117796,62734,-121081,-93041,0
C00874=49427,53549,-117825,62647,-121099,-93060,0
C00875=49580,53533,-117882,62471,-121136,-93099,0
C00876=49732,53517,-117938,62296,-121173,-93137,0
C00877=49746,53516,-117944,62281,-121175,-93141,0
C00878=49759,53514,-117949,62266,-121178,-93144,0
C00879=49772,53512,-117955,62250,-121181,-93148,0
C00880=49785,53511,-117961,62235,-121184,-93152,0
C00881=49798,53509,-117967,62220,-121186,-93155,0
C00882=49811,53507,-117972,62205,-121189,-93159,0
C00883=49824,53506,-117978,62190,-121192,-93162,0
C00884=49837,53504,-117985,62174,-121195,-93166,0
C00885=49850,53502,-117991,62159,-121197,-93170,0
C00886=49863,53501,-117996,62144,-121200,-93173,0
C00887=49876,53499,-118002,62129,-121203,-93177,0
C00888=49889,53497,-118008,62114,-121205,-93180,0
C00889=49901,53495,-118015,62100,-121207,-93184,0
C00890=49913,53493,-118022,62086,-121209,-93188,0
C00891=49925,53492,-118027,62072,-121211,-93191,0
C00892=49937,53490,-118034,62058,-121213,-93195,0
C00893=49948,53488,-118041,62044,-121215,-93198,0
C00894=49959,53486,-118048,62031,-121216,-93202,0
C00895=49970,53484,-118055,62018,-121218,-93206,0
C00896=49981,53481,-118062,62005,-121220,-93209,0
C00897=49992,53479,-118069,61992,-121221,-93213,0
C00898=50003,53477,-118076,61979,-121222,-93216,0
C00899=50014,53475,-118083,61966,-121223,-93220,0
C00900=50025,53473,-118090,61952,-121226,-93224,0
C00901=50033,53472,-118094,61944,-121227,-93226,0
C00902=50044,53470,-118100,61930,-121228,-93230,0
C00903=50055,53468,-118107,61917,-121230,-93233,0
C00904=50067,53467,-118113,61904,-121232,-93236,0
C00905=50073,53466,-118116,61897,-121234,-93238,0
C00906=50084,53459,-118138,61881,-121229,-93246,0
C00907=50110,53444,-118187,61846,-121220,-93263,0
C00908=50138,53428,-118242,61807,-121208,-93283,0
C00909=50166,53411,-118298,61768,-121198,-93303,0
C00910=50189,53396,-118346,61735,-121188,-93320,0
C00911=50208,53384,-118386,61708,-121178,-93334,0
C00912=50227,53372,-118427,61682,-121170,-93348,0
C00913=50242,53361,-118464,61660,-121161,-93360,0
C00914=50258,53350,-118501,61637,-121153,-93372,0
C00915=50273,53339,-118537,61615,-121144,-93385,0
C00916=50288,53328,-118573,61593,-121136,-93397,0
C00917=50303,53317,-118610,61571,-121127,-93410,0
C00918=50315,53307,-118642,61553,-121119,-93421,0
C00919=50327,53298,-118674,61535,-121111,-93432,0
C00920=50340,53288,-118705,61518,-121103,-93442,0
C00921=50352,53278,-118738,61500,-121095,-93453,0
C00922=50361,53270,-118766,61485,-121088,-93462,0
C00923=50371,53261,-118795,61470,-121080,-93472,0
C00924=50381,53253,-118824,61455,-121073,-93481,0
C00925=50390,53244,-118851,61441,-121065,-93490,0
C00926=50400,53236,-118880,61426,-121057,-93500,0
C00927=50410,53227,-118909,61411,-121050,-93509,0
C00928=50419,53218,-118938,61396,-121042,-93518,0
C00929=50428,53211,-118964,61383,-121035,-93527,0
C00930=50436,53203,-118989,61370,-121028,-93535,0
C00931=50444,53195,-119016,61357,-121020,-93544,0
C00932=50442,53191,-119030,61358,-121014,-93547,0
C00933=50435,53182,-119058,61361,-121000,-93554,0
C00934=50430,53174,-119086,61363,-120988,-93561,0
C00935=50423,53165,-119115,61366,-120973,-93568,0
C00936=50416,53155,-119146,61370,-120959,-93576,0
C00937=50409,53146,-119175,61373,-120944,-93583,0
C00938=50402,53137,-119207,61377,-120929,-93590,0
C00939=50395,53127,-119238,61380,-120914,-93598,0
C00940=50388,53118,-119267,61383,-120900,-93605,0
C00941=50380,53109,-119298,61387,-120885,-93613,0
C00942=50372,53099,-119331,61391,-120869,-93620,0
C00943=50363,53089,-119365,61396,-120853,-93629,0
C00944=50354,53078,-119400,61401,-120836,-93637,0
C00945=50345,53068,-119434,61406,-120819,-93645,0
C00946=50334,53057,-119471,61413,-120800,-93654,0
C00947=50322,53044,-119511,61421,-120781,-93663,0
C00948=50310,53032,-119550,61428,-120760,-93672,0
C00949=50298,53020,-119590,61436,-120741,-93682,0
C00950=50285,53008,-119629,61443,-120720,-93691,0
C00951=50272,52996,-119672,61453,-120698,-93700,0
C00952=50256,52982,-119717,61463,-120675,-93711,0
C00953=50241,52969,-119762,61474,-120652,-93721,0
C00954=50219,52951,-119818,61490,-120622,-93733,0
C00955=50197,52934,-119874,61506,-120591,-93746,0
C00956=50175,52917,-119930,61522,-120561,-93758,0
C00957=50168,52915,-119937,61529,-120557,-93759,0
C00958=50159,52913,-119945,61537,-120550,-93760,0
C00959=50148,52910,-119955,61548,-120543,-93761,0
C00960=50137,52907,-119964,61558,-120535,-93762,0
C00961=50127,52904,-119973,61569,-120527,-93764,0
C00962=50116,52901,-119982,61580,-120520,-93764,0
C00963=50105,52898,-119991,61590,-120512,-93765,0
C00964=50094,52896,-120001,61601,-120505,-93766,0
C00965=50082,52893,-120010,61613,-120497,-93767,0
C00966=50070,52890,-120019,61625,-120489,-93768,0
C00967=50058,52887,-120028,61637,-120481,-93769,0
C00968=50045,52884,-120036,61649,-120473,-93769,0
C00969=50033,52881,-120045,61662,-120465,-93770,0
C00970=50021,52879,-120055,61674,-120457,-93771,0
C00971=50009,52876,-120064,61686,-120449,-93772,0
C00972=49996,52873,-120073,61698,-120441,-93772,0
C00973=49984,52870,-120082,61710,-120433,-93773,0
C00974=49972,52867,-120091,61723,-120425,-93774,0
C00975=49960,52865,-120101,61735,-120417,-93775,0
C00976=49947,52862,-120109,61748,-120409,-93775,0
C00977=49933,52859,-120118,61761,-120400,-93776,0
C00978=49920,52857,-120126,61774,-120392,-93776,0
C00979=49906,52854,-120134,61789,-120384,-93776,0
C00980=49891,52851,-120143,61804,-120375,-93777,0
C00981=49875,52849,-120151,61820,-120366,-93777,0
C00982=49860,52846,-120160,61836,-120358,-93777,0
C00983=49844,52843,-120169,61852,-120349,-93777,0
C00984=49829,52840,-120178,61868,-120340,-93777,0
C00985=49813,52838,-120186,61883,-120330,-93777,0
C00986=49801,52835,-120194,61896,-120323,-93778,0
C00987=49723,52821,-120241,61975,-120276,-93780,0
C00988=49578,52794,-120325,62123,-120191,-93783,0
C00989=49432,52768,-120407,62271,-120106,-93786,0
C00990=30265,51930,-122805,60449,-119455,-94584,0
C00991=30178,51866,-123025,60515,-119335,-94634,0
C00992=30092,51803,-123246,60581,-119216,-94684,0
C00993=30044,51769,-123365,60618,-119150,-94711,0
C00994=30036,51763,-123384,60625,-119140,-94715,0
C00995=30027,51758,-123402,60632,-119130,-94719,0
C00996=30019,51752,-123422,60638,-119119,-94724,0
C00997=30011,51747,-123440,60645,-119109,-94728,0
C00998=30002,51741,-123458,60652,-119097,-94732,0
C00999=29994,51736,-123478,60658,-119087,-94736,0
C01000=29986,51731,-123496,60665,-119077,-94740,0
C01001=29977,51725,-123515,60672,-119066,-94744,0
C01002=29969,51720,-123534,60679,-119056,-94749,0
C01003=29961,51715,-123553,60685,-119046,-94753,0
C01004=29953,51710,-123570,60692,-119035,-94756,0
//INST
///DATE 2025/02/20 16:20
///COMM Generated using RoboDK
///ATTR SC,RW
///GROUP1 RB1
NOP
MOVL C00000 V=30.0 PL=1
MOVL C00001 V=30.0 PL=1
MOVL C00002 V=30.0 PL=1
MOVL C00003 V=30.0 PL=1
MOVL C00004 V=30.0 PL=1
MOVL C00005 V=30.0 PL=1
MOVL C00006 V=30.0 PL=1
MOVL C00007 V=30.0 PL=1
MOVL C00008 V=30.0 PL=1
MOVL C00009 V=30.0 PL=1
MOVL C00010 V=30.0 PL=1
MOVL C00011 V=30.0 PL=1
MOVL C00012 V=30.0 PL=1
MOVL C00013 V=30.0 PL=1
MOVL C00014 V=30.0 PL=1
MOVL C00015 V=30.0 PL=1
MOVL C00016 V=30.0 PL=1
MOVL C00017 V=30.0 PL=1
MOVL C00018 V=30.0 PL=1
MOVL C00019 V=30.0 PL=1
MOVL C00020 V=30.0 PL=1
MOVL C00021 V=30.0 PL=1
MOVL C00022 V=30.0 PL=1
MOVL C00023 V=30.0 PL=1
MOVL C00024 V=30.0 PL=1
MOVL C00025 V=30.0 PL=1
MOVL C00026 V=30.0 PL=1
MOVL C00027 V=30.0 PL=1
MOVL C00028 V=30.0 PL=1
MOVL C00029 V=30.0 PL=1
MOVL C00030 V=30.0 PL=1
MOVL C00031 V=30.0 PL=1
MOVL C00032 V=30.0 PL=1
MOVL C00033 V=30.0 PL=1
MOVL C00034 V=30.0 PL=1
MOVL C00035 V=30.0 PL=1
MOVL C00036 V=30.0 PL=1
MOVL C00037 V=30.0 PL=1
MOVL C00038 V=30.0 PL=1
MOVL C00039 V=30.0 PL=1
MOVL C00040 V=30.0 PL=1
MOVL C00041 V=30.0 PL=1
MOVL C00042 V=30.0 PL=1
MOVL C00043 V=30.0 PL=1
MOVL C00044 V=30.0 PL=1
MOVL C00045 V=30.0 PL=1
MOVL C00046 V=30.0 PL=1
MOVL C00047 V=30.0 PL=1
MOVL C00048 V=30.0 PL=1
MOVL C00049 V=30.0 PL=1
MOVL C00050 V=30.0 PL=1
MOVL C00051 V=30.0 PL=1
MOVL C00052 V=30.0 PL=1
MOVL C00053 V=30.0 PL=1
MOVL C00054 V=30.0 PL=1
MOVL C00055 V=30.0 PL=1
MOVL C00056 V=30.0 PL=1
MOVL C00057 V=30.0 PL=1
MOVL C00058 V=30.0 PL=1
MOVL C00059 V=30.0 PL=1
MOVL C00060 V=30.0 PL=1
MOVL C00061 V=30.0 PL=1
MOVL C00062 V=30.0 PL=1
MOVL C00063 V=30.0 PL=1
MOVL C00064 V=30.0 PL=1
MOVL C00065 V=30.0 PL=1
MOVL C00066 V=30.0 PL=1
MOVL C00067 V=30.0 PL=1
MOVL C00068 V=30.0 PL=1
MOVL C00069 V=30.0 PL=1
MOVL C00070 V=30.0 PL=1
MOVL C00071 V=30.0 PL=1
MOVL C00072 V=30.0 PL=1
MOVL C00073 V=30.0 PL=1
MOVL C00074 V=30.0 PL=1
MOVL C00075 V=30.0 PL=1
MOVL C00076 V=30.0 PL=1
MOVL C00077 V=30.0 PL=1
MOVL C00078 V=30.0 PL=1
MOVL C00079 V=30.0 PL=1
MOVL C00080 V=30.0 PL=1
MOVL C00081 V=30.0 PL=1
MOVL C00082 V=30.0 PL=1
MOVL C00083 V=30.0 PL=1
MOVL C00084 V=30.0 PL=1
MOVL C00085 V=30.0 PL=1
MOVL C00086 V=30.0 PL=1
MOVL C00087 V=30.0 PL=1
MOVL C00088 V=30.0 PL=1
MOVL C00089 V=30.0 PL=1
MOVL C00090 V=30.0 PL=1
MOVL C00091 V=30.0 PL=1
MOVL C00092 V=30.0 PL=1
MOVL C00093 V=30.0 PL=1
MOVL C00094 V=30.0 PL=1
MOVL C00095 V=30.0 PL=1
MOVL C00096 V=30.0 PL=1
MOVL C00097 V=30.0 PL=1
MOVL C00098 V=30.0 PL=1
MOVL C00099 V=30.0 PL=1
MOVL C00100 V=130.0 PL=1
MOVL C00101 V=80.0 PL=1
MOVL C00102 V=130.0 PL=1
MOVL C00103 V=80.0 PL=1
MOVL C00104 V=130.0 PL=1
MOVL C00105 V=80.0 PL=1
MOVL C00106 V=130.0 PL=1
MOVL C00107 V=80.0 PL=1
MOVL C00108 V=80.0 PL=1
MOVL C00109 V=80.0 PL=1
MOVL C00110 V=80.0 PL=1
MOVL C00111 V=80.0 PL=1
MOVL C00112 V=80.0 PL=1
MOVL C00113 V=80.0 PL=1
MOVL C00114 V=80.0 PL=1
MOVL C00115 V=80.0 PL=1
MOVL C00116 V=80.0 PL=1
MOVL C00117 V=80.0 PL=1
MOVL C00118 V=130.0 PL=1
MOVL C00119 V=130.0 PL=1
MOVL C00120 V=60.0 PL=1
MOVL C00121 V=60.0 PL=1
MOVL C00122 V=60.0 PL=1
MOVL C00123 V=60.0 PL=1
MOVL C00124 V=60.0 PL=1
MOVL C00125 V=60.0 PL=1
MOVL C00126 V=60.0 PL=1
MOVL C00127 V=60.0 PL=1
MOVL C00128 V=60.0 PL=1
MOVL C00129 V=60.0 PL=1
MOVL C00130 V=60.0 PL=1
MOVL C00131 V=60.0 PL=1
MOVL C00132 V=60.0 PL=1
MOVL C00133 V=60.0 PL=1
MOVL C00134 V=60.0 PL=1
MOVL C00135 V=60.0 PL=1
MOVL C00136 V=60.0 PL=1
MOVL C00137 V=60.0 PL=1
MOVL C00138 V=60.0 PL=1
MOVL C00139 V=60.0 PL=1
MOVL C00140 V=60.0 PL=1
MOVL C00141 V=60.0 PL=1
MOVL C00142 V=60.0 PL=1
MOVL C00143 V=60.0 PL=1
MOVL C00144 V=130.0 PL=1
MOVL C00145 V=60.0 PL=1
MOVL C00146 V=60.0 PL=1
MOVL C00147 V=60.0 PL=1
MOVL C00148 V=60.0 PL=1
MOVL C00149 V=60.0 PL=1
MOVL C00150 V=60.0 PL=1
MOVL C00151 V=60.0 PL=1
MOVL C00152 V=60.0 PL=1
MOVL C00153 V=60.0 PL=1
MOVL C00154 V=60.0 PL=1
MOVL C00155 V=60.0 PL=1
MOVL C00156 V=60.0 PL=1
MOVL C00157 V=60.0 PL=1
MOVL C00158 V=60.0 PL=1
MOVL C00159 V=60.0 PL=1
MOVL C00160 V=60.0 PL=1
MOVL C00161 V=60.0 PL=1
MOVL C00162 V=60.0 PL=1
MOVL C00163 V=60.0 PL=1
MOVL C00164 V=60.0 PL=1
MOVL C00165 V=60.0 PL=1
MOVL C00166 V=60.0 PL=1
MOVL C00167 V=60.0 PL=1
MOVL C00168 V=60.0 PL=1
MOVL C00169 V=60.0 PL=1
MOVL C00170 V=60.0 PL=1
MOVL C00171 V=60.0 PL=1
MOVL C00172 V=60.0 PL=1
MOVL C00173 V=60.0 PL=1
MOVL C00174 V=60.0 PL=1
MOVL C00175 V=60.0 PL=1
MOVL C00176 V=60.0 PL=1
MOVL C00177 V=60.0 PL=1
MOVL C00178 V=60.0 PL=1
MOVL C00179 V=60.0 PL=1
MOVL C00180 V=60.0 PL=1
MOVL C00181 V=60.0 PL=1
MOVL C00182 V=60.0 PL=1
MOVL C00183 V=60.0 PL=1
MOVL C00184 V=60.0 PL=1
MOVL C00185 V=130.0 PL=1
MOVL C00186 V=30.0 PL=1
MOVL C00187 V=30.0 PL=1
MOVL C00188 V=30.0 PL=1
MOVL C00189 V=30.0 PL=1
MOVL C00190 V=30.0 PL=1
MOVL C00191 V=30.0 PL=1
MOVL C00192 V=30.0 PL=1
MOVL C00193 V=30.0 PL=1
MOVL C00194 V=30.0 PL=1
MOVL C00195 V=30.0 PL=1
MOVL C00196 V=30.0 PL=1
MOVL C00197 V=30.0 PL=1
MOVL C00198 V=30.0 PL=1
MOVL C00199 V=30.0 PL=1
MOVL C00200 V=30.0 PL=1
MOVL C00201 V=30.0 PL=1
MOVL C00202 V=30.0 PL=1
MOVL C00203 V=30.0 PL=1
MOVL C00204 V=30.0 PL=1
MOVL C00205 V=30.0 PL=1
MOVL C00206 V=30.0 PL=1
MOVL C00207 V=30.0 PL=1
MOVL C00208 V=30.0 PL=1
MOVL C00209 V=30.0 PL=1
MOVL C00210 V=30.0 PL=1
MOVL C00211 V=30.0 PL=1
MOVL C00212 V=30.0 PL=1
MOVL C00213 V=30.0 PL=1
MOVL C00214 V=30.0 PL=1
MOVL C00215 V=30.0 PL=1
MOVL C00216 V=30.0 PL=1
MOVL C00217 V=30.0 PL=1
MOVL C00218 V=30.0 PL=1
MOVL C00219 V=30.0 PL=1
MOVL C00220 V=30.0 PL=1
MOVL C00221 V=30.0 PL=1
MOVL C00222 V=30.0 PL=1
MOVL C00223 V=30.0 PL=1
MOVL C00224 V=30.0 PL=1
MOVL C00225 V=30.0 PL=1
MOVL C00226 V=30.0 PL=1
MOVL C00227 V=30.0 PL=1
MOVL C00228 V=30.0 PL=1
MOVL C00229 V=30.0 PL=1
MOVL C00230 V=30.0 PL=1
MOVL C00231 V=30.0 PL=1
MOVL C00232 V=30.0 PL=1
MOVL C00233 V=30.0 PL=1
MOVL C00234 V=30.0 PL=1
MOVL C00235 V=30.0 PL=1
MOVL C00236 V=30.0 PL=1
MOVL C00237 V=30.0 PL=1
MOVL C00238 V=30.0 PL=1
MOVL C00239 V=30.0 PL=1
MOVL C00240 V=30.0 PL=1
MOVL C00241 V=30.0 PL=1
MOVL C00242 V=30.0 PL=1
MOVL C00243 V=30.0 PL=1
MOVL C00244 V=30.0 PL=1
MOVL C00245 V=30.0 PL=1
MOVL C00246 V=30.0 PL=1
MOVL C00247 V=30.0 PL=1
MOVL C00248 V=30.0 PL=1
MOVL C00249 V=30.0 PL=1
MOVL C00250 V=30.0 PL=1
MOVL C00251 V=30.0 PL=1
MOVL C00252 V=30.0 PL=1
MOVL C00253 V=30.0 PL=1
MOVL C00254 V=30.0 PL=1
MOVL C00255 V=30.0 PL=1
MOVL C00256 V=30.0 PL=1
MOVL C00257 V=30.0 PL=1
MOVL C00258 V=130.0 PL=1
MOVL C00259 V=130.0 PL=1
MOVL C00260 V=30.0 PL=1
MOVL C00261 V=30.0 PL=1
MOVL C00262 V=30.0 PL=1
MOVL C00263 V=30.0 PL=1
MOVL C00264 V=30.0 PL=1
MOVL C00265 V=30.0 PL=1
MOVL C00266 V=30.0 PL=1
MOVL C00267 V=30.0 PL=1
MOVL C00268 V=30.0 PL=1
MOVL C00269 V=30.0 PL=1
MOVL C00270 V=30.0 PL=1
MOVL C00271 V=30.0 PL=1
MOVL C00272 V=30.0 PL=1
MOVL C00273 V=30.0 PL=1
MOVL C00274 V=30.0 PL=1
MOVL C00275 V=30.0 PL=1
MOVL C00276 V=30.0 PL=1
MOVL C00277 V=30.0 PL=1
MOVL C00278 V=30.0 PL=1
MOVL C00279 V=30.0 PL=1
MOVL C00280 V=30.0 PL=1
MOVL C00281 V=30.0 PL=1
MOVL C00282 V=30.0 PL=1
MOVL C00283 V=30.0 PL=1
MOVL C00284 V=30.0 PL=1
MOVL C00285 V=30.0 PL=1
MOVL C00286 V=30.0 PL=1
MOVL C00287 V=30.0 PL=1
MOVL C00288 V=30.0 PL=1
MOVL C00289 V=30.0 PL=1
MOVL C00290 V=30.0 PL=1
MOVL C00291 V=30.0 PL=1
MOVL C00292 V=30.0 PL=1
MOVL C00293 V=30.0 PL=1
MOVL C00294 V=30.0 PL=1
MOVL C00295 V=30.0 PL=1
MOVL C00296 V=30.0 PL=1
MOVL C00297 V=30.0 PL=1
MOVL C00298 V=30.0 PL=1
MOVL C00299 V=30.0 PL=1
MOVL C00300 V=30.0 PL=1
MOVL C00301 V=30.0 PL=1
MOVL C00302 V=30.0 PL=1
MOVL C00303 V=30.0 PL=1
MOVL C00304 V=30.0 PL=1
MOVL C00305 V=30.0 PL=1
MOVL C00306 V=30.0 PL=1
MOVL C00307 V=30.0 PL=1
MOVL C00308 V=30.0 PL=1
MOVL C00309 V=30.0 PL=1
MOVL C00310 V=30.0 PL=1
MOVL C00311 V=30.0 PL=1
MOVL C00312 V=30.0 PL=1
MOVL C00313 V=30.0 PL=1
MOVL C00314 V=30.0 PL=1
MOVL C00315 V=30.0 PL=1
MOVL C00316 V=30.0 PL=1
MOVL C00317 V=30.0 PL=1
MOVL C00318 V=30.0 PL=1
MOVL C00319 V=30.0 PL=1
MOVL C00320 V=30.0 PL=1
MOVL C00321 V=30.0 PL=1
MOVL C00322 V=30.0 PL=1
MOVL C00323 V=30.0 PL=1
MOVL C00324 V=30.0 PL=1
MOVL C00325 V=30.0 PL=1
MOVL C00326 V=30.0 PL=1
MOVL C00327 V=30.0 PL=1
MOVL C00328 V=30.0 PL=1
MOVL C00329 V=30.0 PL=1
MOVL C00330 V=30.0 PL=1
MOVL C00331 V=30.0 PL=1
MOVL C00332 V=30.0 PL=1
MOVL C00333 V=30.0 PL=1
MOVL C00334 V=30.0 PL=1
MOVL C00335 V=30.0 PL=1
MOVL C00336 V=30.0 PL=1
MOVL C00337 V=30.0 PL=1
MOVL C00338 V=30.0 PL=1
MOVL C00339 V=30.0 PL=1
MOVL C00340 V=30.0 PL=1
MOVL C00341 V=30.0 PL=1
MOVL C00342 V=30.0 PL=1
MOVL C00343 V=30.0 PL=1
MOVL C00344 V=30.0 PL=1
MOVL C00345 V=30.0 PL=1
MOVL C00346 V=30.0 PL=1
MOVL C00347 V=30.0 PL=1
MOVL C00348 V=30.0 PL=1
MOVL C00349 V=30.0 PL=1
MOVL C00350 V=30.0 PL=1
MOVL C00351 V=30.0 PL=1
MOVL C00352 V=30.0 PL=1
MOVL C00353 V=30.0 PL=1
MOVL C00354 V=30.0 PL=1
MOVL C00355 V=30.0 PL=1
MOVL C00356 V=30.0 PL=1
MOVL C00357 V=30.0 PL=1
MOVL C00358 V=30.0 PL=1
MOVL C00359 V=30.0 PL=1
MOVL C00360 V=30.0 PL=1
MOVL C00361 V=30.0 PL=1
MOVL C00362 V=130.0 PL=1
MOVL C00363 V=30.0 PL=1
MOVL C00364 V=30.0 PL=1
MOVL C00365 V=30.0 PL=1
MOVL C00366 V=30.0 PL=1
MOVL C00367 V=30.0 PL=1
MOVL C00368 V=30.0 PL=1
MOVL C00369 V=30.0 PL=1
MOVL C00370 V=30.0 PL=1
MOVL C00371 V=30.0 PL=1
MOVL C00372 V=30.0 PL=1
MOVL C00373 V=30.0 PL=1
MOVL C00374 V=30.0 PL=1
MOVL C00375 V=30.0 PL=1
MOVL C00376 V=30.0 PL=1
MOVL C00377 V=30.0 PL=1
MOVL C00378 V=30.0 PL=1
MOVL C00379 V=30.0 PL=1
MOVL C00380 V=30.0 PL=1
MOVL C00381 V=30.0 PL=1
MOVL C00382 V=30.0 PL=1
MOVL C00383 V=30.0 PL=1
MOVL C00384 V=30.0 PL=1
MOVL C00385 V=30.0 PL=1
MOVL C00386 V=30.0 PL=1
MOVL C00387 V=30.0 PL=1
MOVL C00388 V=30.0 PL=1
MOVL C00389 V=30.0 PL=1
MOVL C00390 V=30.0 PL=1
MOVL C00391 V=30.0 PL=1
MOVL C00392 V=30.0 PL=1
MOVL C00393 V=30.0 PL=1
MOVL C00394 V=30.0 PL=1
MOVL C00395 V=30.0 PL=1
MOVL C00396 V=30.0 PL=1
MOVL C00397 V=30.0 PL=1
MOVL C00398 V=30.0 PL=1
MOVL C00399 V=30.0 PL=1
MOVL C00400 V=30.0 PL=1
MOVL C00401 V=30.0 PL=1
MOVL C00402 V=30.0 PL=1
MOVL C00403 V=30.0 PL=1
MOVL C00404 V=30.0 PL=1
MOVL C00405 V=30.0 PL=1
MOVL C00406 V=30.0 PL=1
MOVL C00407 V=30.0 PL=1
MOVL C00408 V=30.0 PL=1
MOVL C00409 V=30.0 PL=1
MOVL C00410 V=30.0 PL=1
MOVL C00411 V=30.0 PL=1
MOVL C00412 V=30.0 PL=1
MOVL C00413 V=30.0 PL=1
MOVL C00414 V=30.0 PL=1
MOVL C00415 V=30.0 PL=1
MOVL C00416 V=30.0 PL=1
MOVL C00417 V=30.0 PL=1
MOVL C00418 V=30.0 PL=1
MOVL C00419 V=30.0 PL=1
MOVL C00420 V=30.0 PL=1
MOVL C00421 V=30.0 PL=1
MOVL C00422 V=30.0 PL=1
MOVL C00423 V=30.0 PL=1
MOVL C00424 V=30.0 PL=1
MOVL C00425 V=30.0 PL=1
MOVL C00426 V=30.0 PL=1
MOVL C00427 V=30.0 PL=1
MOVL C00428 V=30.0 PL=1
MOVL C00429 V=30.0 PL=1
MOVL C00430 V=30.0 PL=1
MOVL C00431 V=30.0 PL=1
MOVL C00432 V=30.0 PL=1
MOVL C00433 V=30.0 PL=1
MOVL C00434 V=30.0 PL=1
MOVL C00435 V=30.0 PL=1
MOVL C00436 V=30.0 PL=1
MOVL C00437 V=30.0 PL=1
MOVL C00438 V=30.0 PL=1
MOVL C00439 V=30.0 PL=1
MOVL C00440 V=30.0 PL=1
MOVL C00441 V=30.0 PL=1
MOVL C00442 V=30.0 PL=1
MOVL C00443 V=30.0 PL=1
MOVL C00444 V=30.0 PL=1
MOVL C00445 V=30.0 PL=1
MOVL C00446 V=30.0 PL=1
MOVL C00447 V=30.0 PL=1
MOVL C00448 V=30.0 PL=1
MOVL C00449 V=30.0 PL=1
MOVL C00450 V=30.0 PL=1
MOVL C00451 V=30.0 PL=1
MOVL C00452 V=30.0 PL=1
MOVL C00453 V=30.0 PL=1
MOVL C00454 V=30.0 PL=1
MOVL C00455 V=30.0 PL=1
MOVL C00456 V=30.0 PL=1
MOVL C00457 V=30.0 PL=1
MOVL C00458 V=30.0 PL=1
MOVL C00459 V=30.0 PL=1
MOVL C00460 V=30.0 PL=1
MOVL C00461 V=30.0 PL=1
MOVL C00462 V=30.0 PL=1
MOVL C00463 V=30.0 PL=1
MOVL C00464 V=30.0 PL=1
MOVL C00465 V=30.0 PL=1
MOVL C00466 V=30.0 PL=1
MOVL C00467 V=130.0 PL=1
MOVL C00468 V=30.0 PL=1
MOVL C00469 V=30.0 PL=1
MOVL C00470 V=30.0 PL=1
MOVL C00471 V=30.0 PL=1
MOVL C00472 V=30.0 PL=1
MOVL C00473 V=30.0 PL=1
MOVL C00474 V=30.0 PL=1
MOVL C00475 V=30.0 PL=1
MOVL C00476 V=30.0 PL=1
MOVL C00477 V=30.0 PL=1
MOVL C00478 V=30.0 PL=1
MOVL C00479 V=30.0 PL=1
MOVL C00480 V=30.0 PL=1
MOVL C00481 V=30.0 PL=1
MOVL C00482 V=30.0 PL=1
MOVL C00483 V=30.0 PL=1
MOVL C00484 V=30.0 PL=1
MOVL C00485 V=30.0 PL=1
MOVL C00486 V=30.0 PL=1
MOVL C00487 V=30.0 PL=1
MOVL C00488 V=30.0 PL=1
MOVL C00489 V=30.0 PL=1
MOVL C00490 V=30.0 PL=1
MOVL C00491 V=30.0 PL=1
MOVL C00492 V=30.0 PL=1
MOVL C00493 V=30.0 PL=1
MOVL C00494 V=30.0 PL=1
MOVL C00495 V=30.0 PL=1
MOVL C00496 V=30.0 PL=1
MOVL C00497 V=30.0 PL=1
MOVL C00498 V=30.0 PL=1
MOVL C00499 V=30.0 PL=1
MOVL C00500 V=30.0 PL=1
MOVL C00501 V=30.0 PL=1
MOVL C00502 V=30.0 PL=1
MOVL C00503 V=30.0 PL=1
MOVL C00504 V=30.0 PL=1
MOVL C00505 V=30.0 PL=1
MOVL C00506 V=30.0 PL=1
MOVL C00507 V=30.0 PL=1
MOVL C00508 V=30.0 PL=1
MOVL C00509 V=30.0 PL=1
MOVL C00510 V=30.0 PL=1
MOVL C00511 V=30.0 PL=1
MOVL C00512 V=30.0 PL=1
MOVL C00513 V=30.0 PL=1
MOVL C00514 V=30.0 PL=1
MOVL C00515 V=30.0 PL=1
MOVL C00516 V=30.0 PL=1
MOVL C00517 V=30.0 PL=1
MOVL C00518 V=30.0 PL=1
MOVL C00519 V=30.0 PL=1
MOVL C00520 V=30.0 PL=1
MOVL C00521 V=30.0 PL=1
MOVL C00522 V=30.0 PL=1
MOVL C00523 V=30.0 PL=1
MOVL C00524 V=30.0 PL=1
MOVL C00525 V=30.0 PL=1
MOVL C00526 V=30.0 PL=1
MOVL C00527 V=30.0 PL=1
MOVL C00528 V=30.0 PL=1
MOVL C00529 V=30.0 PL=1
MOVL C00530 V=30.0 PL=1
MOVL C00531 V=30.0 PL=1
MOVL C00532 V=30.0 PL=1
MOVL C00533 V=30.0 PL=1
MOVL C00534 V=30.0 PL=1
MOVL C00535 V=30.0 PL=1
MOVL C00536 V=30.0 PL=1
MOVL C00537 V=30.0 PL=1
MOVL C00538 V=30.0 PL=1
MOVL C00539 V=30.0 PL=1
MOVL C00540 V=30.0 PL=1
MOVL C00541 V=30.0 PL=1
MOVL C00542 V=30.0 PL=1
MOVL C00543 V=30.0 PL=1
MOVL C00544 V=30.0 PL=1
MOVL C00545 V=30.0 PL=1
MOVL C00546 V=30.0 PL=1
MOVL C00547 V=30.0 PL=1
MOVL C00548 V=30.0 PL=1
MOVL C00549 V=30.0 PL=1
MOVL C00550 V=30.0 PL=1
MOVL C00551 V=30.0 PL=1
MOVL C00552 V=30.0 PL=1
MOVL C00553 V=30.0 PL=1
MOVL C00554 V=30.0 PL=1
MOVL C00555 V=30.0 PL=1
MOVL C00556 V=30.0 PL=1
MOVL C00557 V=30.0 PL=1
MOVL C00558 V=30.0 PL=1
MOVL C00559 V=30.0 PL=1
MOVL C00560 V=30.0 PL=1
MOVL C00561 V=30.0 PL=1
MOVL C00562 V=30.0 PL=1
MOVL C00563 V=30.0 PL=1
MOVL C00564 V=30.0 PL=1
MOVL C00565 V=30.0 PL=1
MOVL C00566 V=30.0 PL=1
MOVL C00567 V=30.0 PL=1
MOVL C00568 V=30.0 PL=1
MOVL C00569 V=30.0 PL=1
MOVL C00570 V=30.0 PL=1
MOVL C00571 V=30.0 PL=1
MOVL C00572 V=30.0 PL=1
MOVL C00573 V=30.0 PL=1
MOVL C00574 V=30.0 PL=1
MOVL C00575 V=30.0 PL=1
MOVL C00576 V=30.0 PL=1
MOVL C00577 V=30.0 PL=1
MOVL C00578 V=30.0 PL=1
MOVL C00579 V=30.0 PL=1
MOVL C00580 V=30.0 PL=1
MOVL C00581 V=30.0 PL=1
MOVL C00582 V=30.0 PL=1
MOVL C00583 V=30.0 PL=1
MOVL C00584 V=30.0 PL=1
MOVL C00585 V=130.0 PL=1
MOVL C00586 V=30.0 PL=1
MOVL C00587 V=30.0 PL=1
MOVL C00588 V=30.0 PL=1
MOVL C00589 V=30.0 PL=1
MOVL C00590 V=30.0 PL=1
MOVL C00591 V=30.0 PL=1
MOVL C00592 V=30.0 PL=1
MOVL C00593 V=30.0 PL=1
MOVL C00594 V=30.0 PL=1
MOVL C00595 V=30.0 PL=1
MOVL C00596 V=30.0 PL=1
MOVL C00597 V=30.0 PL=1
MOVL C00598 V=30.0 PL=1
MOVL C00599 V=30.0 PL=1
MOVL C00600 V=30.0 PL=1
MOVL C00601 V=30.0 PL=1
MOVL C00602 V=30.0 PL=1
MOVL C00603 V=30.0 PL=1
MOVL C00604 V=30.0 PL=1
MOVL C00605 V=30.0 PL=1
MOVL C00606 V=30.0 PL=1
MOVL C00607 V=30.0 PL=1
MOVL C00608 V=30.0 PL=1
MOVL C00609 V=30.0 PL=1
MOVL C00610 V=30.0 PL=1
MOVL C00611 V=30.0 PL=1
MOVL C00612 V=30.0 PL=1
MOVL C00613 V=30.0 PL=1
MOVL C00614 V=30.0 PL=1
MOVL C00615 V=30.0 PL=1
MOVL C00616 V=30.0 PL=1
MOVL C00617 V=30.0 PL=1
MOVL C00618 V=30.0 PL=1
MOVL C00619 V=30.0 PL=1
MOVL C00620 V=30.0 PL=1
MOVL C00621 V=30.0 PL=1
MOVL C00622 V=30.0 PL=1
MOVL C00623 V=30.0 PL=1
MOVL C00624 V=30.0 PL=1
MOVL C00625 V=30.0 PL=1
MOVL C00626 V=30.0 PL=1
MOVL C00627 V=30.0 PL=1
MOVL C00628 V=30.0 PL=1
MOVL C00629 V=30.0 PL=1
MOVL C00630 V=30.0 PL=1
MOVL C00631 V=30.0 PL=1
MOVL C00632 V=30.0 PL=1
MOVL C00633 V=30.0 PL=1
MOVL C00634 V=30.0 PL=1
MOVL C00635 V=30.0 PL=1
MOVL C00636 V=30.0 PL=1
MOVL C00637 V=30.0 PL=1
MOVL C00638 V=30.0 PL=1
MOVL C00639 V=30.0 PL=1
MOVL C00640 V=30.0 PL=1
MOVL C00641 V=30.0 PL=1
MOVL C00642 V=30.0 PL=1
MOVL C00643 V=30.0 PL=1
MOVL C00644 V=30.0 PL=1
MOVL C00645 V=30.0 PL=1
MOVL C00646 V=30.0 PL=1
MOVL C00647 V=30.0 PL=1
MOVL C00648 V=30.0 PL=1
MOVL C00649 V=30.0 PL=1
MOVL C00650 V=30.0 PL=1
MOVL C00651 V=30.0 PL=1
MOVL C00652 V=30.0 PL=1
MOVL C00653 V=30.0 PL=1
MOVL C00654 V=30.0 PL=1
MOVL C00655 V=30.0 PL=1
MOVL C00656 V=30.0 PL=1
MOVL C00657 V=30.0 PL=1
MOVL C00658 V=30.0 PL=1
MOVL C00659 V=30.0 PL=1
MOVL C00660 V=30.0 PL=1
MOVL C00661 V=30.0 PL=1
MOVL C00662 V=30.0 PL=1
MOVL C00663 V=30.0 PL=1
MOVL C00664 V=30.0 PL=1
MOVL C00665 V=30.0 PL=1
MOVL C00666 V=30.0 PL=1
MOVL C00667 V=30.0 PL=1
MOVL C00668 V=30.0 PL=1
MOVL C00669 V=30.0 PL=1
MOVL C00670 V=30.0 PL=1
MOVL C00671 V=30.0 PL=1
MOVL C00672 V=30.0 PL=1
MOVL C00673 V=30.0 PL=1
MOVL C00674 V=30.0 PL=1
MOVL C00675 V=30.0 PL=1
MOVL C00676 V=30.0 PL=1
MOVL C00677 V=30.0 PL=1
MOVL C00678 V=30.0 PL=1
MOVL C00679 V=30.0 PL=1
MOVL C00680 V=30.0 PL=1
MOVL C00681 V=30.0 PL=1
MOVL C00682 V=30.0 PL=1
MOVL C00683 V=30.0 PL=1
MOVL C00684 V=30.0 PL=1
MOVL C00685 V=30.0 PL=1
MOVL C00686 V=30.0 PL=1
MOVL C00687 V=30.0 PL=1
MOVL C00688 V=30.0 PL=1
MOVL C00689 V=30.0 PL=1
MOVL C00690 V=30.0 PL=1
MOVL C00691 V=30.0 PL=1
MOVL C00692 V=30.0 PL=1
MOVL C00693 V=30.0 PL=1
MOVL C00694 V=30.0 PL=1
MOVL C00695 V=30.0 PL=1
MOVL C00696 V=30.0 PL=1
MOVL C00697 V=30.0 PL=1
MOVL C00698 V=30.0 PL=1
MOVL C00699 V=30.0 PL=1
MOVL C00700 V=30.0 PL=1
MOVL C00701 V=30.0 PL=1
MOVL C00702 V=30.0 PL=1
MOVL C00703 V=130.0 PL=1
MOVL C00704 V=80.0 PL=1
MOVL C00705 V=130.0 PL=1
MOVL C00706 V=80.0 PL=1
MOVL C00707 V=130.0 PL=1
MOVL C00708 V=80.0 PL=1
MOVL C00709 V=130.0 PL=1
MOVL C00710 V=80.0 PL=1
MOVL C00711 V=80.0 PL=1
MOVL C00712 V=80.0 PL=1
MOVL C00713 V=80.0 PL=1
MOVL C00714 V=80.0 PL=1
MOVL C00715 V=80.0 PL=1
MOVL C00716 V=80.0 PL=1
MOVL C00717 V=80.0 PL=1
MOVL C00718 V=80.0 PL=1
MOVL C00719 V=80.0 PL=1
MOVL C00720 V=80.0 PL=1
MOVL C00721 V=80.0 PL=1
MOVL C00722 V=80.0 PL=1
MOVL C00723 V=80.0 PL=1
MOVL C00724 V=130.0 PL=1
MOVL C00725 V=130.0 PL=1
MOVL C00726 V=60.0 PL=1
MOVL C00727 V=60.0 PL=1
MOVL C00728 V=60.0 PL=1
MOVL C00729 V=60.0 PL=1
MOVL C00730 V=60.0 PL=1
MOVL C00731 V=60.0 PL=1
MOVL C00732 V=60.0 PL=1
MOVL C00733 V=60.0 PL=1
MOVL C00734 V=60.0 PL=1
MOVL C00735 V=60.0 PL=1
MOVL C00736 V=60.0 PL=1
MOVL C00737 V=60.0 PL=1
MOVL C00738 V=60.0 PL=1
MOVL C00739 V=60.0 PL=1
MOVL C00740 V=60.0 PL=1
MOVL C00741 V=60.0 PL=1
MOVL C00742 V=60.0 PL=1
MOVL C00743 V=60.0 PL=1
MOVL C00744 V=60.0 PL=1
MOVL C00745 V=60.0 PL=1
MOVL C00746 V=60.0 PL=1
MOVL C00747 V=60.0 PL=1
MOVL C00748 V=60.0 PL=1
MOVL C00749 V=60.0 PL=1
MOVL C00750 V=60.0 PL=1
MOVL C00751 V=60.0 PL=1
MOVL C00752 V=60.0 PL=1
MOVL C00753 V=60.0 PL=1
MOVL C00754 V=130.0 PL=1
MOVL C00755 V=60.0 PL=1
MOVL C00756 V=60.0 PL=1
MOVL C00757 V=60.0 PL=1
MOVL C00758 V=60.0 PL=1
MOVL C00759 V=60.0 PL=1
MOVL C00760 V=60.0 PL=1
MOVL C00761 V=60.0 PL=1
MOVL C00762 V=60.0 PL=1
MOVL C00763 V=60.0 PL=1
MOVL C00764 V=60.0 PL=1
MOVL C00765 V=60.0 PL=1
MOVL C00766 V=60.0 PL=1
MOVL C00767 V=60.0 PL=1
MOVL C00768 V=60.0 PL=1
MOVL C00769 V=60.0 PL=1
MOVL C00770 V=60.0 PL=1
MOVL C00771 V=60.0 PL=1
MOVL C00772 V=60.0 PL=1
MOVL C00773 V=60.0 PL=1
MOVL C00774 V=60.0 PL=1
MOVL C00775 V=60.0 PL=1
MOVL C00776 V=60.0 PL=1
MOVL C00777 V=60.0 PL=1
MOVL C00778 V=60.0 PL=1
MOVL C00779 V=60.0 PL=1
MOVL C00780 V=60.0 PL=1
MOVL C00781 V=60.0 PL=1
MOVL C00782 V=60.0 PL=1
MOVL C00783 V=60.0 PL=1
MOVL C00784 V=60.0 PL=1
MOVL C00785 V=60.0 PL=1
MOVL C00786 V=60.0 PL=1
MOVL C00787 V=60.0 PL=1
MOVL C00788 V=60.0 PL=1
MOVL C00789 V=60.0 PL=1
MOVL C00790 V=60.0 PL=1
MOVL C00791 V=60.0 PL=1
MOVL C00792 V=60.0 PL=1
MOVL C00793 V=60.0 PL=1
MOVL C00794 V=60.0 PL=1
MOVL C00795 V=60.0 PL=1
MOVL C00796 V=60.0 PL=1
MOVL C00797 V=60.0 PL=1
MOVL C00798 V=60.0 PL=1
MOVL C00799 V=130.0 PL=1
MOVL C00800 V=30.0 PL=1
MOVL C00801 V=30.0 PL=1
MOVL C00802 V=30.0 PL=1
MOVL C00803 V=30.0 PL=1
MOVL C00804 V=30.0 PL=1
MOVL C00805 V=30.0 PL=1
MOVL C00806 V=30.0 PL=1
MOVL C00807 V=30.0 PL=1
MOVL C00808 V=30.0 PL=1
MOVL C00809 V=30.0 PL=1
MOVL C00810 V=30.0 PL=1
MOVL C00811 V=30.0 PL=1
MOVL C00812 V=30.0 PL=1
MOVL C00813 V=30.0 PL=1
MOVL C00814 V=30.0 PL=1
MOVL C00815 V=30.0 PL=1
MOVL C00816 V=30.0 PL=1
MOVL C00817 V=30.0 PL=1
MOVL C00818 V=30.0 PL=1
MOVL C00819 V=30.0 PL=1
MOVL C00820 V=30.0 PL=1
MOVL C00821 V=30.0 PL=1
MOVL C00822 V=30.0 PL=1
MOVL C00823 V=30.0 PL=1
MOVL C00824 V=30.0 PL=1
MOVL C00825 V=30.0 PL=1
MOVL C00826 V=30.0 PL=1
MOVL C00827 V=30.0 PL=1
MOVL C00828 V=30.0 PL=1
MOVL C00829 V=30.0 PL=1
MOVL C00830 V=30.0 PL=1
MOVL C00831 V=30.0 PL=1
MOVL C00832 V=30.0 PL=1
MOVL C00833 V=30.0 PL=1
MOVL C00834 V=30.0 PL=1
MOVL C00835 V=30.0 PL=1
MOVL C00836 V=30.0 PL=1
MOVL C00837 V=30.0 PL=1
MOVL C00838 V=30.0 PL=1
MOVL C00839 V=30.0 PL=1
MOVL C00840 V=30.0 PL=1
MOVL C00841 V=30.0 PL=1
MOVL C00842 V=30.0 PL=1
MOVL C00843 V=30.0 PL=1
MOVL C00844 V=30.0 PL=1
MOVL C00845 V=30.0 PL=1
MOVL C00846 V=30.0 PL=1
MOVL C00847 V=30.0 PL=1
MOVL C00848 V=30.0 PL=1
MOVL C00849 V=30.0 PL=1
MOVL C00850 V=30.0 PL=1
MOVL C00851 V=30.0 PL=1
MOVL C00852 V=30.0 PL=1
MOVL C00853 V=30.0 PL=1
MOVL C00854 V=30.0 PL=1
MOVL C00855 V=30.0 PL=1
MOVL C00856 V=30.0 PL=1
MOVL C00857 V=30.0 PL=1
MOVL C00858 V=30.0 PL=1
MOVL C00859 V=30.0 PL=1
MOVL C00860 V=30.0 PL=1
MOVL C00861 V=30.0 PL=1
MOVL C00862 V=30.0 PL=1
MOVL C00863 V=30.0 PL=1
MOVL C00864 V=30.0 PL=1
MOVL C00865 V=30.0 PL=1
MOVL C00866 V=30.0 PL=1
MOVL C00867 V=30.0 PL=1
MOVL C00868 V=30.0 PL=1
MOVL C00869 V=30.0 PL=1
MOVL C00870 V=30.0 PL=1
MOVL C00871 V=30.0 PL=1
MOVL C00872 V=130.0 PL=1
MOVL C00873 V=130.0 PL=1
MOVL C00874 V=30.0 PL=1
MOVL C00875 V=30.0 PL=1
MOVL C00876 V=30.0 PL=1
MOVL C00877 V=30.0 PL=1
MOVL C00878 V=30.0 PL=1
MOVL C00879 V=30.0 PL=1
MOVL C00880 V=30.0 PL=1
MOVL C00881 V=30.0 PL=1
MOVL C00882 V=30.0 PL=1
MOVL C00883 V=30.0 PL=1
MOVL C00884 V=30.0 PL=1
MOVL C00885 V=30.0 PL=1
MOVL C00886 V=30.0 PL=1
MOVL C00887 V=30.0 PL=1
MOVL C00888 V=30.0 PL=1
MOVL C00889 V=30.0 PL=1
MOVL C00890 V=30.0 PL=1
MOVL C00891 V=30.0 PL=1
MOVL C00892 V=30.0 PL=1
MOVL C00893 V=30.0 PL=1
MOVL C00894 V=30.0 PL=1
MOVL C00895 V=30.0 PL=1
MOVL C00896 V=30.0 PL=1
MOVL C00897 V=30.0 PL=1
MOVL C00898 V=30.0 PL=1
MOVL C00899 V=30.0 PL=1
MOVL C00900 V=30.0 PL=1
MOVL C00901 V=30.0 PL=1
MOVL C00902 V=30.0 PL=1
MOVL C00903 V=30.0 PL=1
MOVL C00904 V=30.0 PL=1
MOVL C00905 V=30.0 PL=1
MOVL C00906 V=30.0 PL=1
MOVL C00907 V=30.0 PL=1
MOVL C00908 V=30.0 PL=1
MOVL C00909 V=30.0 PL=1
MOVL C00910 V=30.0 PL=1
MOVL C00911 V=30.0 PL=1
MOVL C00912 V=30.0 PL=1
MOVL C00913 V=30.0 PL=1
MOVL C00914 V=30.0 PL=1
MOVL C00915 V=30.0 PL=1
MOVL C00916 V=30.0 PL=1
MOVL C00917 V=30.0 PL=1
MOVL C00918 V=30.0 PL=1
MOVL C00919 V=30.0 PL=1
MOVL C00920 V=30.0 PL=1
MOVL C00921 V=30.0 PL=1
MOVL C00922 V=30.0 PL=1
MOVL C00923 V=30.0 PL=1
MOVL C00924 V=30.0 PL=1
MOVL C00925 V=30.0 PL=1
MOVL C00926 V=30.0 PL=1
MOVL C00927 V=30.0 PL=1
MOVL C00928 V=30.0 PL=1
MOVL C00929 V=30.0 PL=1
MOVL C00930 V=30.0 PL=1
MOVL C00931 V=30.0 PL=1
MOVL C00932 V=30.0 PL=1
MOVL C00933 V=30.0 PL=1
MOVL C00934 V=30.0 PL=1
MOVL C00935 V=30.0 PL=1
MOVL C00936 V=30.0 PL=1
MOVL C00937 V=30.0 PL=1
MOVL C00938 V=30.0 PL=1
MOVL C00939 V=30.0 PL=1
MOVL C00940 V=30.0 PL=1
MOVL C00941 V=30.0 PL=1
MOVL C00942 V=30.0 PL=1
MOVL C00943 V=30.0 PL=1
MOVL C00944 V=30.0 PL=1
MOVL C00945 V=30.0 PL=1
MOVL C00946 V=30.0 PL=1
MOVL C00947 V=30.0 PL=1
MOVL C00948 V=30.0 PL=1
MOVL C00949 V=30.0 PL=1
MOVL C00950 V=30.0 PL=1
MOVL C00951 V=30.0 PL=1
MOVL C00952 V=30.0 PL=1
MOVL C00953 V=30.0 PL=1
MOVL C00954 V=30.0 PL=1
MOVL C00955 V=30.0 PL=1
MOVL C00956 V=30.0 PL=1
MOVL C00957 V=30.0 PL=1
MOVL C00958 V=30.0 PL=1
MOVL C00959 V=30.0 PL=1
MOVL C00960 V=30.0 PL=1
MOVL C00961 V=30.0 PL=1
MOVL C00962 V=30.0 PL=1
MOVL C00963 V=30.0 PL=1
MOVL C00964 V=30.0 PL=1
MOVL C00965 V=30.0 PL=1
MOVL C00966 V=30.0 PL=1
MOVL C00967 V=30.0 PL=1
MOVL C00968 V=30.0 PL=1
MOVL C00969 V=30.0 PL=1
MOVL C00970 V=30.0 PL=1
MOVL C00971 V=30.0 PL=1
MOVL C00972 V=30.0 PL=1
MOVL C00973 V=30.0 PL=1
MOVL C00974 V=30.0 PL=1
MOVL C00975 V=30.0 PL=1
MOVL C00976 V=30.0 PL=1
MOVL C00977 V=30.0 PL=1
MOVL C00978 V=30.0 PL=1
MOVL C00979 V=30.0 PL=1
MOVL C00980 V=30.0 PL=1
MOVL C00981 V=30.0 PL=1
MOVL C00982 V=30.0 PL=1
MOVL C00983 V=30.0 PL=1
MOVL C00984 V=30.0 PL=1
MOVL C00985 V=30.0 PL=1
MOVL C00986 V=30.0 PL=1
MOVL C00987 V=30.0 PL=1
MOVL C00988 V=30.0 PL=1
MOVL C00989 V=30.0 PL=1
MOVL C00990 V=130.0 PL=1
MOVL C00991 V=30.0 PL=1
MOVL C00992 V=30.0 PL=1
MOVL C00993 V=30.0 PL=1
MOVL C00994 V=30.0 PL=1
MOVL C00995 V=30.0 PL=1
MOVL C00996 V=30.0 PL=1
MOVL C00997 V=30.0 PL=1
MOVL C00998 V=30.0 PL=1
MOVL C00999 V=30.0 PL=1
MOVL C01000 V=30.0 PL=1
MOVL C01001 V=30.0 PL=1
MOVL C01002 V=30.0 PL=1
MOVL C01003 V=30.0 PL=1
MOVL C01004 V=30.0 PL=1
END
